LIN {X 0,Y 573.266,Z 445.075,A -85,B 0,C 180,E1 -2313.81,E2 -2313.81} C_VEL
LIN {X 0,Y 573.234,Z 445.082,A -85,B 0,C 180,E1 -2316.135,E2 -2316.135} C_VEL
LIN {X 0,Y 573.254,Z 445.079,A -85,B 0,C 180,E1 -2319.174,E2 -2319.174} C_VEL
LIN {X 0,Y 573.23,Z 445.081,A -85,B 0,C 180,E1 -2321.412,E2 -2321.412} C_VEL
LIN {X 0,Y 573.254,Z 445.077,A -85,B 0,C 180,E1 -2323.622,E2 -2323.622} C_VEL
LIN {X 0,Y 573.276,Z 445.079,A -85,B 0,C 180,E1 -2325.807,E2 -2325.807} C_VEL
LIN {X 0,Y 573.266,Z 445.08,A -85,B 0,C 180,E1 -2328.745,E2 -2328.745} C_VEL
LIN {X 0,Y 573.287,Z 445.073,A -85,B 0,C 180,E1 -2331.541,E2 -2331.541} C_VEL
LIN {X 0,Y 573.292,Z 445.072,A -85,B 0,C 180,E1 -2334.372,E2 -2334.372} C_VEL
LIN {X 0,Y 573.308,Z 445.071,A -85,B 0,C 180,E1 -2337.893,E2 -2337.893} C_VEL
LIN {X 0,Y 573.337,Z 445.066,A -85,B 0,C 180,E1 -2340.702,E2 -2340.702} C_VEL
LIN {X 0,Y 573.234,Z 445.079,A -85,B 0,C 180,E1 -2343.515,E2 -2343.515} C_VEL
LIN {X 0,Y 573.291,Z 445.073,A -85,B 0,C 180,E1 -2345.628,E2 -2345.628} C_VEL
LIN {X 0,Y 573.292,Z 445.072,A -85,B 0,C 180,E1 -2348.46,E2 -2348.46} C_VEL
LIN {X 0,Y 573.275,Z 445.073,A -85,B 0,C 180,E1 -2351.312,E2 -2351.312} C_VEL
LIN {X 0,Y 573.285,Z 445.073,A -85,B 0,C 180,E1 -2354.425,E2 -2354.425} C_VEL
LIN {X 0,Y 573.262,Z 445.079,A -85,B 0,C 180,E1 -2357.112,E2 -2357.112} C_VEL
LIN {X 0,Y 573.255,Z 445.082,A -85,B 0,C 180,E1 -2360.077,E2 -2360.077} C_VEL
LIN {X 0,Y 573.238,Z 445.084,A -85,B 0,C 180,E1 -2363.1,E2 -2363.1} C_VEL
LIN {X 0,Y 573.253,Z 445.079,A -85,B 0,C 180,E1 -2364.389,E2 -2364.389} C_VEL
LIN {X 0,Y 572.625,Z 445.161,A -85,B 0,C 180,E1 -2364.976,E2 -2364.976} C_VEL
LIN {X 0,Y 569.778,Z 445.516,A -85,B 0,C 180,E1 -2365.927,E2 -2365.927} C_VEL
LIN {X 0,Y 567.345,Z 445.816,A -85,B 0,C 180,E1 -2366.692,E2 -2366.692} C_VEL
LIN {X 0,Y 566.296,Z 445.944,A -85,B 0,C 180,E1 -2367.284,E2 -2367.284} C_VEL
LIN {X 0,Y 566.21,Z 445.954,A -85,B 0,C 180,E1 -2367.484,E2 -2367.484} C_VEL
LIN {X 0,Y 566.205,Z 445.957,A -85,B 0,C 180,E1 -2369.769,E2 -2369.769} C_VEL
LIN {X 0,Y 566.209,Z 445.959,A -85,B 0,C 180,E1 -2372.43,E2 -2372.43} C_VEL
LIN {X 0,Y 566.205,Z 445.955,A -85,B 0,C 180,E1 -2374.993,E2 -2374.993} C_VEL
LIN {X 0,Y 566.2,Z 445.958,A -85,B 0,C 180,E1 -2377.461,E2 -2377.461} C_VEL
LIN {X 0,Y 566.21,Z 445.958,A -85,B 0,C 180,E1 -2380.199,E2 -2380.199} C_VEL
LIN {X 0,Y 566.209,Z 445.956,A -85,B 0,C 180,E1 -2383.054,E2 -2383.054} C_VEL
LIN {X 0,Y 566.202,Z 445.956,A -85,B 0,C 180,E1 -2386.049,E2 -2386.049} C_VEL
LIN {X 0,Y 566.207,Z 445.955,A -85,B 0,C 180,E1 -2389.215,E2 -2389.215} C_VEL
LIN {X 0,Y 566.19,Z 445.958,A -85,B 0,C 180,E1 -2391.637,E2 -2391.637} C_VEL
LIN {X 0,Y 566.196,Z 445.961,A -85,B 0,C 180,E1 -2394.31,E2 -2394.31} C_VEL
LIN {X 0,Y 566.224,Z 445.952,A -85,B 0,C 180,E1 -2396.898,E2 -2396.898} C_VEL
LIN {X 0,Y 566.184,Z 445.959,A -85,B 0,C 180,E1 -2399.407,E2 -2399.407} C_VEL
LIN {X 0,Y 566.199,Z 445.957,A -85,B 0,C 180,E1 -2401.857,E2 -2401.857} C_VEL
LIN {X 0,Y 566.218,Z 445.954,A -85,B 0,C 180,E1 -2404.251,E2 -2404.251} C_VEL
LIN {X 0,Y 566.178,Z 445.963,A -85,B 0,C 180,E1 -2406.718,E2 -2406.718} C_VEL
LIN {X 0,Y 566.211,Z 445.956,A -85,B 0,C 180,E1 -2409.663,E2 -2409.663} C_VEL
LIN {X 0,Y 566.204,Z 445.956,A -85,B 0,C 180,E1 -2412.669,E2 -2412.669} C_VEL
LIN {X 0,Y 566.24,Z 445.95,A -85,B 0,C 180,E1 -2415.627,E2 -2415.627} C_VEL
LIN {X 0,Y 566.241,Z 445.95,A -85,B 0,C 180,E1 -2418.675,E2 -2418.675} C_VEL
LIN {X 0,Y 566.233,Z 445.952,A -85,B 0,C 180,E1 -2421.434,E2 -2421.434} C_VEL
LIN {X 0,Y 566.257,Z 445.95,A -85,B 0,C 180,E1 -2424.302,E2 -2424.302} C_VEL
LIN {X 0,Y 566.288,Z 445.944,A -85,B 0,C 180,E1 -2427.866,E2 -2427.866} C_VEL
LIN {X 0,Y 566.304,Z 445.943,A -85,B 0,C 180,E1 -2430.711,E2 -2430.711} C_VEL
LIN {X 0,Y 566.273,Z 445.947,A -85,B 0,C 180,E1 -2432.846,E2 -2432.846} C_VEL
LIN {X 0,Y 566.263,Z 445.947,A -85,B 0,C 180,E1 -2435.698,E2 -2435.698} C_VEL
LIN {X 0,Y 566.212,Z 445.954,A -85,B 0,C 180,E1 -2438.566,E2 -2438.566} C_VEL
LIN {X 0,Y 566.248,Z 445.952,A -85,B 0,C 180,E1 -2441.454,E2 -2441.454} C_VEL
LIN {X 0,Y 566.241,Z 445.953,A -85,B 0,C 180,E1 -2444.507,E2 -2444.507} C_VEL
LIN {X 0,Y 566.205,Z 445.959,A -85,B 0,C 180,E1 -2447.332,E2 -2447.332} C_VEL
LIN {X 0,Y 566.214,Z 445.957,A -85,B 0,C 180,E1 -2450.337,E2 -2450.337} C_VEL
LIN {X 0,Y 566.178,Z 445.959,A -85,B 0,C 180,E1 -2453.282,E2 -2453.282} C_VEL
LIN {X 0,Y 566.219,Z 445.953,A -85,B 0,C 180,E1 -2455.749,E2 -2455.749} C_VEL
LIN {X 0,Y 566.208,Z 445.959,A -85,B 0,C 180,E1 -2458.202,E2 -2458.202} C_VEL
LIN {X 0,Y 566.196,Z 445.957,A -85,B 0,C 180,E1 -2461.076,E2 -2461.076} C_VEL
LIN {X 0,Y 566.217,Z 445.953,A -85,B 0,C 180,E1 -2463.734,E2 -2463.734} C_VEL
LIN {X 0,Y 566.204,Z 445.955,A -85,B 0,C 180,E1 -2466.57,E2 -2466.57} C_VEL
LIN {X 0,Y 566.225,Z 445.953,A -85,B 0,C 180,E1 -2469.686,E2 -2469.686} C_VEL
LIN {X 0,Y 566.216,Z 445.956,A -85,B 0,C 180,E1 -2472.087,E2 -2472.087} C_VEL
LIN {X 0,Y 566.174,Z 445.959,A -85,B 0,C 180,E1 -2475.036,E2 -2475.036} C_VEL
LIN {X 0,Y 566.223,Z 445.954,A -85,B 0,C 180,E1 -2478.136,E2 -2478.136} C_VEL
LIN {X 0,Y 566.216,Z 445.953,A -85,B 0,C 180,E1 -2480.726,E2 -2480.726} C_VEL
LIN {X 0,Y 566.197,Z 445.96,A -85,B 0,C 180,E1 -2483.429,E2 -2483.429} C_VEL
LIN {X 0,Y 566.027,Z 445.982,A -85,B 0,C 180,E1 -2486.031,E2 -2486.031} C_VEL
LIN {X 0,Y 565.995,Z 446.653,A -85,B 0,C 180,E1 -2486.883,E2 -2486.883} C_VEL
LIN {X 0,Y 565.971,Z 449.517,A -85,B 0,C 180,E1 -2489.394,E2 -2489.394} C_VEL
LIN {X 0,Y 565.965,Z 452.327,A -85,B 0,C 180,E1 -2491.844,E2 -2491.844} C_VEL
LIN {X 0,Y 565.945,Z 455.14,A -85,B 0,C 180,E1 -2494.238,E2 -2494.238} C_VEL
LIN {X 0,Y 565.898,Z 458.02,A -85,B 0,C 180,E1 -2496.784,E2 -2496.784} C_VEL
LIN {X 0,Y 565.884,Z 461.612,A -85,B 0,C 180,E1 -2499.65,E2 -2499.65} C_VEL
LIN {X 0,Y 565.864,Z 465.455,A -85,B 0,C 180,E1 -2502.658,E2 -2502.658} C_VEL
LIN {X 0,Y 565.889,Z 469.316,A -85,B 0,C 180,E1 -2505.631,E2 -2505.631} C_VEL
LIN {X 0,Y 565.897,Z 471.671,A -85,B 0,C 180,E1 -2507.424,E2 -2507.424} C_VEL
LIN {X 0,Y 566.89,Z 479.272,A -85,B 0,C 180,E1 -2507.629,E2 -2507.629} C_VEL
LIN {X 0,Y 566.784,Z 491.774,A -85,B 0,C 180,E1 -2508.013,E2 -2508.013} C_VEL
LIN {X 0,Y 566.661,Z 504.296,A -85,B 0,C 180,E1 -2508.554,E2 -2508.554} C_VEL
LIN {X 0,Y 566.544,Z 515.576,A -85,B 0,C 180,E1 -2509.192,E2 -2509.192} C_VEL
LIN {X 0,Y 566.342,Z 526.839,A -85,B 0,C 180,E1 -2509.995,E2 -2509.995} C_VEL
LIN {X 0,Y 566.238,Z 536.889,A -85,B 0,C 180,E1 -2510.895,E2 -2510.895} C_VEL
LIN {X 0,Y 566.113,Z 546.59,A -85,B 0,C 180,E1 -2511.971,E2 -2511.971} C_VEL
LIN {X 0,Y 566.05,Z 553.158,A -85,B 0,C 180,E1 -2512.868,E2 -2512.868} C_VEL
LIN {X 0,Y 566.003,Z 559.627,A -85,B 0,C 180,E1 -2513.941,E2 -2513.941} C_VEL
LIN {X 0,Y 565.878,Z 564.764,A -85,B 0,C 180,E1 -2515.012,E2 -2515.012} C_VEL
LIN {X 0,Y 565.926,Z 568.753,A -85,B 0,C 180,E1 -2516.083,E2 -2516.083} C_VEL
LIN {X 0,Y 565.878,Z 571.701,A -85,B 0,C 180,E1 -2517.152,E2 -2517.152} C_VEL
LIN {X 0,Y 565.839,Z 573.128,A -85,B 0,C 180,E1 -2517.864,E2 -2517.864} C_VEL
LIN {X 0,Y 565.842,Z 574.756,A -85,B 0,C 180,E1 -2519.288,E2 -2519.288} C_VEL
LIN {X 0,Y 565.839,Z 574.996,A -85,B 0,C 180,E1 -2520,E2 -2520} C_VEL
LIN {X 0,Y 565.841,Z 574.815,A -85,B 0,C 180,E1 -2520.712,E2 -2520.712} C_VEL
LIN {X 0,Y 565.838,Z 573.269,A -85,B 0,C 180,E1 -2522.135,E2 -2522.135} C_VEL
LIN {X 0,Y 565.878,Z 571.908,A -85,B 0,C 180,E1 -2522.847,E2 -2522.847} C_VEL
LIN {X 0,Y 565.926,Z 569.03,A -85,B 0,C 180,E1 -2523.916,E2 -2523.916} C_VEL
LIN {X 0,Y 565.878,Z 565.13,A -85,B 0,C 180,E1 -2524.987,E2 -2524.987} C_VEL
LIN {X 0,Y 565.994,Z 560.097,A -85,B 0,C 180,E1 -2526.058,E2 -2526.058} C_VEL
LIN {X 0,Y 566.031,Z 553.773,A -85,B 0,C 180,E1 -2527.132,E2 -2527.132} C_VEL
LIN {X 0,Y 566.128,Z 545.851,A -85,B 0,C 180,E1 -2528.208,E2 -2528.208} C_VEL
LIN {X 0,Y 566.249,Z 536,A -85,B 0,C 180,E1 -2529.285,E2 -2529.285} C_VEL
LIN {X 0,Y 566.412,Z 525.679,A -85,B 0,C 180,E1 -2530.184,E2 -2530.184} C_VEL
LIN {X 0,Y 566.525,Z 514.433,A -85,B 0,C 180,E1 -2530.97,E2 -2530.97} C_VEL
LIN {X 0,Y 566.684,Z 502.858,A -85,B 0,C 180,E1 -2531.608,E2 -2531.608} C_VEL
LIN {X 0,Y 566.783,Z 490.466,A -85,B 0,C 180,E1 -2532.124,E2 -2532.124} C_VEL
LIN {X 0,Y 566.817,Z 477.42,A -85,B 0,C 180,E1 -2532.509,E2 -2532.509} C_VEL
LIN {X 0,Y 565.899,Z 471.67,A -85,B 0,C 180,E1 -2532.666,E2 -2532.666} C_VEL
LIN {X 0,Y 565.857,Z 468.455,A -85,B 0,C 180,E1 -2535.119,E2 -2535.119} C_VEL
LIN {X 0,Y 565.863,Z 465.571,A -85,B 0,C 180,E1 -2537.342,E2 -2537.342} C_VEL
LIN {X 0,Y 565.884,Z 461.726,A -85,B 0,C 180,E1 -2540.35,E2 -2540.35} C_VEL
LIN {X 0,Y 565.898,Z 458.134,A -85,B 0,C 180,E1 -2543.216,E2 -2543.216} C_VEL
LIN {X 0,Y 565.962,Z 455.534,A -85,B 0,C 180,E1 -2545.761,E2 -2545.761} C_VEL
LIN {X 0,Y 566.028,Z 453.112,A -85,B 0,C 180,E1 -2548.168,E2 -2548.168} C_VEL
LIN {X 0,Y 566.078,Z 450.089,A -85,B 0,C 180,E1 -2551.057,E2 -2551.057} C_VEL
LIN {X 0,Y 566.109,Z 447.052,A -85,B 0,C 180,E1 -2553.963,E2 -2553.963} C_VEL
LIN {X 0,Y 566.117,Z 446.004,A -85,B 0,C 180,E1 -2554.98,E2 -2554.98} C_VEL
LIN {X 0,Y 566.2,Z 445.959,A -85,B 0,C 180,E1 -2557.461,E2 -2557.461} C_VEL
LIN {X 0,Y 566.21,Z 445.96,A -85,B 0,C 180,E1 -2560.199,E2 -2560.199} C_VEL
LIN {X 0,Y 566.209,Z 445.958,A -85,B 0,C 180,E1 -2563.054,E2 -2563.054} C_VEL
LIN {X 0,Y 566.201,Z 445.96,A -85,B 0,C 180,E1 -2566.049,E2 -2566.049} C_VEL
LIN {X 0,Y 566.224,Z 445.956,A -85,B 0,C 180,E1 -2569.212,E2 -2569.212} C_VEL
LIN {X 0,Y 566.209,Z 445.959,A -85,B 0,C 180,E1 -2572.091,E2 -2572.091} C_VEL
LIN {X 0,Y 566.225,Z 446.171,A -85,B 0,C 180,E1 -2572.596,E2 -2572.596} C_VEL
LIN {X 0,Y 566.879,Z 450.21,A -85,B 0,C 180,E1 -2574.36,E2 -2574.36} C_VEL
LIN {X 0,Y 566.688,Z 456.223,A -85,B 0,C 180,E1 -2576.553,E2 -2576.553} C_VEL
LIN {X 0,Y 566.562,Z 463.236,A -85,B 0,C 180,E1 -2578.862,E2 -2578.862} C_VEL
LIN {X 0,Y 566.448,Z 471.711,A -85,B 0,C 180,E1 -2581.443,E2 -2581.443} C_VEL
LIN {X 0,Y 566.425,Z 480.069,A -85,B 0,C 180,E1 -2583.866,E2 -2583.866} C_VEL
LIN {X 0,Y 566.361,Z 488.309,A -85,B 0,C 180,E1 -2586.216,E2 -2586.216} C_VEL
LIN {X 0,Y 566.245,Z 497.576,A -85,B 0,C 180,E1 -2588.904,E2 -2588.904} C_VEL
LIN {X 0,Y 566.167,Z 506.844,A -85,B 0,C 180,E1 -2591.546,E2 -2591.546} C_VEL
LIN {X 0,Y 566.092,Z 517.435,A -85,B 0,C 180,E1 -2594.519,E2 -2594.519} C_VEL
LIN {X 0,Y 566.033,Z 527.53,A -85,B 0,C 180,E1 -2597.314,E2 -2597.314} C_VEL
LIN {X 0,Y 566.942,Z 534.363,A -85,B 0,C 180,E1 -2597.471,E2 -2597.471} C_VEL
LIN {X 0,Y 566.829,Z 546.495,A -85,B 0,C 180,E1 -2597.786,E2 -2597.786} C_VEL
LIN {X 0,Y 566.719,Z 558.314,A -85,B 0,C 180,E1 -2598.229,E2 -2598.229} C_VEL
LIN {X 0,Y 566.572,Z 570.724,A -85,B 0,C 180,E1 -2598.854,E2 -2598.854} C_VEL
LIN {X 0,Y 566.419,Z 581.48,A -85,B 0,C 180,E1 -2599.545,E2 -2599.545} C_VEL
LIN {X 0,Y 566.301,Z 591.646,A -85,B 0,C 180,E1 -2600.355,E2 -2600.355} C_VEL
LIN {X 0,Y 566.166,Z 600.786,A -85,B 0,C 180,E1 -2601.253,E2 -2601.253} C_VEL
LIN {X 0,Y 566.08,Z 609.689,A -85,B 0,C 180,E1 -2602.33,E2 -2602.33} C_VEL
LIN {X 0,Y 565.967,Z 616.955,A -85,B 0,C 180,E1 -2603.422,E2 -2603.422} C_VEL
LIN {X 0,Y 566.004,Z 621.679,A -85,B 0,C 180,E1 -2604.299,E2 -2604.299} C_VEL
LIN {X 0,Y 565.933,Z 626.372,A -85,B 0,C 180,E1 -2605.37,E2 -2605.37} C_VEL
LIN {X 0,Y 565.927,Z 629.957,A -85,B 0,C 180,E1 -2606.44,E2 -2606.44} C_VEL
LIN {X 0,Y 565.878,Z 631.808,A -85,B 0,C 180,E1 -2607.152,E2 -2607.152} C_VEL
LIN {X 0,Y 565.846,Z 634.186,A -85,B 0,C 180,E1 -2608.577,E2 -2608.577} C_VEL
LIN {X 0,Y 565.839,Z 635,A -85,B 0,C 180,E1 -2610,E2 -2610} C_VEL
LIN {X 0,Y 565.846,Z 634.186,A -85,B 0,C 180,E1 -2611.423,E2 -2611.423} C_VEL
LIN {X 0,Y 565.878,Z 631.81,A -85,B 0,C 180,E1 -2612.847,E2 -2612.847} C_VEL
LIN {X 0,Y 565.926,Z 628.896,A -85,B 0,C 180,E1 -2613.916,E2 -2613.916} C_VEL
LIN {X 0,Y 565.878,Z 624.949,A -85,B 0,C 180,E1 -2614.987,E2 -2614.987} C_VEL
LIN {X 0,Y 566.002,Z 619.867,A -85,B 0,C 180,E1 -2616.058,E2 -2616.058} C_VEL
LIN {X 0,Y 566.04,Z 613.469,A -85,B 0,C 180,E1 -2617.132,E2 -2617.132} C_VEL
LIN {X 0,Y 566.133,Z 605.479,A -85,B 0,C 180,E1 -2618.208,E2 -2618.208} C_VEL
LIN {X 0,Y 566.229,Z 597.336,A -85,B 0,C 180,E1 -2619.105,E2 -2619.105} C_VEL
LIN {X 0,Y 566.342,Z 587.401,A -85,B 0,C 180,E1 -2620.005,E2 -2620.005} C_VEL
LIN {X 0,Y 566.534,Z 576.299,A -85,B 0,C 180,E1 -2620.807,E2 -2620.807} C_VEL
LIN {X 0,Y 566.612,Z 565.178,A -85,B 0,C 180,E1 -2621.447,E2 -2621.447} C_VEL
LIN {X 0,Y 566.756,Z 552.985,A -85,B 0,C 180,E1 -2621.988,E2 -2621.988} C_VEL
LIN {X 0,Y 566.881,Z 540.178,A -85,B 0,C 180,E1 -2622.394,E2 -2622.394} C_VEL
LIN {X 0,Y 566.716,Z 531.802,A -85,B 0,C 180,E1 -2622.585,E2 -2622.585} C_VEL
LIN {X 0,Y 566.033,Z 527.53,A -85,B 0,C 180,E1 -2622.686,E2 -2622.686} C_VEL
LIN {X 0,Y 566.091,Z 517.436,A -85,B 0,C 180,E1 -2625.481,E2 -2625.481} C_VEL
LIN {X 0,Y 566.167,Z 506.844,A -85,B 0,C 180,E1 -2628.454,E2 -2628.454} C_VEL
LIN {X 0,Y 566.245,Z 497.577,A -85,B 0,C 180,E1 -2631.096,E2 -2631.096} C_VEL
LIN {X 0,Y 566.362,Z 488.31,A -85,B 0,C 180,E1 -2633.784,E2 -2633.784} C_VEL
LIN {X 0,Y 566.473,Z 478.959,A -85,B 0,C 180,E1 -2636.528,E2 -2636.528} C_VEL
LIN {X 0,Y 566.558,Z 469.563,A -85,B 0,C 180,E1 -2639.34,E2 -2639.34} C_VEL
LIN {X 0,Y 566.669,Z 461.593,A -85,B 0,C 180,E1 -2641.81,E2 -2641.81} C_VEL
LIN {X 0,Y 566.865,Z 453.765,A -85,B 0,C 180,E1 -2644.341,E2 -2644.341} C_VEL
LIN {X 0,Y 566.815,Z 449.857,A -85,B 0,C 180,E1 -2645.645,E2 -2645.645} C_VEL
LIN {X 0,Y 566.221,Z 445.957,A -85,B 0,C 180,E1 -2647.061,E2 -2647.061} C_VEL
LIN {X 0,Y 566.215,Z 445.958,A -85,B 0,C 180,E1 -2649.685,E2 -2649.685} C_VEL
LIN {X 0,Y 566.192,Z 445.957,A -85,B 0,C 180,E1 -2652.089,E2 -2652.089} C_VEL
LIN {X 0,Y 566.176,Z 445.959,A -85,B 0,C 180,E1 -2655.036,E2 -2655.036} C_VEL
LIN {X 0,Y 566.217,Z 445.956,A -85,B 0,C 180,E1 -2657.913,E2 -2657.913} C_VEL
LIN {X 0,Y 566.214,Z 445.959,A -85,B 0,C 180,E1 -2660.726,E2 -2660.726} C_VEL
LIN {X 0,Y 566.188,Z 445.962,A -85,B 0,C 180,E1 -2663.788,E2 -2663.788} C_VEL
LIN {X 0,Y 566.214,Z 445.953,A -85,B 0,C 180,E1 -2666.266,E2 -2666.266} C_VEL
LIN {X 0,Y 566.193,Z 445.958,A -85,B 0,C 180,E1 -2668.924,E2 -2668.924} C_VEL
LIN {X 0,Y 566.214,Z 445.958,A -85,B 0,C 180,E1 -2671.857,E2 -2671.857} C_VEL
LIN {X 0,Y 566.216,Z 445.954,A -85,B 0,C 180,E1 -2674.251,E2 -2674.251} C_VEL
LIN {X 0,Y 566.175,Z 445.96,A -85,B 0,C 180,E1 -2676.718,E2 -2676.718} C_VEL
LIN {X 0,Y 566.217,Z 445.957,A -85,B 0,C 180,E1 -2679.663,E2 -2679.663} C_VEL
LIN {X 0,Y 566.202,Z 445.96,A -85,B 0,C 180,E1 -2682.668,E2 -2682.668} C_VEL
LIN {X 0,Y 566.237,Z 445.955,A -85,B 0,C 180,E1 -2685.627,E2 -2685.627} C_VEL
LIN {X 0,Y 566.237,Z 445.954,A -85,B 0,C 180,E1 -2688.675,E2 -2688.675} C_VEL
LIN {X 0,Y 566.23,Z 445.952,A -85,B 0,C 180,E1 -2691.434,E2 -2691.434} C_VEL
LIN {X 0,Y 566.26,Z 445.948,A -85,B 0,C 180,E1 -2694.302,E2 -2694.302} C_VEL
LIN {X 0,Y 566.28,Z 445.947,A -85,B 0,C 180,E1 -2697.866,E2 -2697.866} C_VEL
LIN {X 0,Y 566.307,Z 445.942,A -85,B 0,C 180,E1 -2700.711,E2 -2700.711} C_VEL
LIN {X 0,Y 566.278,Z 445.951,A -85,B 0,C 180,E1 -2702.846,E2 -2702.846} C_VEL
LIN {X 0,Y 566.26,Z 445.95,A -85,B 0,C 180,E1 -2705.698,E2 -2705.698} C_VEL
LIN {X 0,Y 566.236,Z 445.951,A -85,B 0,C 180,E1 -2708.566,E2 -2708.566} C_VEL
LIN {X 0,Y 566.245,Z 445.949,A -85,B 0,C 180,E1 -2711.454,E2 -2711.454} C_VEL
LIN {X 0,Y 566.238,Z 445.951,A -85,B 0,C 180,E1 -2714.507,E2 -2714.507} C_VEL
LIN {X 0,Y 566.203,Z 445.956,A -85,B 0,C 180,E1 -2717.332,E2 -2717.332} C_VEL
LIN {X 0,Y 566.217,Z 445.956,A -85,B 0,C 180,E1 -2720.337,E2 -2720.337} C_VEL
LIN {X 0,Y 566.176,Z 445.963,A -85,B 0,C 180,E1 -2723.282,E2 -2723.282} C_VEL
LIN {X 0,Y 566.216,Z 445.953,A -85,B 0,C 180,E1 -2725.749,E2 -2725.749} C_VEL
LIN {X 0,Y 566.21,Z 445.954,A -85,B 0,C 180,E1 -2727.484,E2 -2727.484} C_VEL
LIN {X 0,Y 565.538,Z 446.041,A -85,B 0,C 180,E1 -2728.078,E2 -2728.078} C_VEL
LIN {X 0,Y 562.671,Z 446.397,A -85,B 0,C 180,E1 -2729.041,E2 -2729.041} C_VEL
LIN {X 0,Y 560.254,Z 446.698,A -85,B 0,C 180,E1 -2729.817,E2 -2729.817} C_VEL
LIN {X 0,Y 559.224,Z 446.825,A -85,B 0,C 180,E1 -2730.415,E2 -2730.415} C_VEL
LIN {X 0,Y 559.143,Z 446.835,A -85,B 0,C 180,E1 -2730.618,E2 -2730.618} C_VEL
LIN {X 0,Y 559.168,Z 446.831,A -85,B 0,C 180,E1 -2733.575,E2 -2733.575} C_VEL
LIN {X 0,Y 559.171,Z 446.831,A -85,B 0,C 180,E1 -2736.448,E2 -2736.448} C_VEL
LIN {X 0,Y 559.177,Z 446.834,A -85,B 0,C 180,E1 -2738.934,E2 -2738.934} C_VEL
LIN {X 0,Y 559.181,Z 446.833,A -85,B 0,C 180,E1 -2742.138,E2 -2742.138} C_VEL
LIN {X 0,Y 559.145,Z 446.837,A -85,B 0,C 180,E1 -2744.739,E2 -2744.739} C_VEL
LIN {X 0,Y 559.161,Z 446.832,A -85,B 0,C 180,E1 -2747.256,E2 -2747.256} C_VEL
LIN {X 0,Y 559.184,Z 446.831,A -85,B 0,C 180,E1 -2750.135,E2 -2750.135} C_VEL
LIN {X 0,Y 559.148,Z 446.838,A -85,B 0,C 180,E1 -2752.892,E2 -2752.892} C_VEL
LIN {X 0,Y 559.172,Z 446.835,A -85,B 0,C 180,E1 -2756.051,E2 -2756.051} C_VEL
LIN {X 0,Y 559.159,Z 446.837,A -85,B 0,C 180,E1 -2758.981,E2 -2758.981} C_VEL
LIN {X 0,Y 559.173,Z 446.831,A -85,B 0,C 180,E1 -2761.619,E2 -2761.619} C_VEL
LIN {X 0,Y 559.181,Z 446.83,A -85,B 0,C 180,E1 -2764.702,E2 -2764.702} C_VEL
LIN {X 0,Y 559.145,Z 446.835,A -85,B 0,C 180,E1 -2767.847,E2 -2767.847} C_VEL
LIN {X 0,Y 559.197,Z 446.828,A -85,B 0,C 180,E1 -2770.494,E2 -2770.494} C_VEL
LIN {X 0,Y 559.184,Z 446.834,A -85,B 0,C 180,E1 -2773.198,E2 -2773.198} C_VEL
LIN {X 0,Y 559.177,Z 446.836,A -85,B 0,C 180,E1 -2776.184,E2 -2776.184} C_VEL
LIN {X 0,Y 559.201,Z 446.831,A -85,B 0,C 180,E1 -2779.134,E2 -2779.134} C_VEL
LIN {X 0,Y 559.209,Z 446.828,A -85,B 0,C 180,E1 -2782.054,E2 -2782.054} C_VEL
LIN {X 0,Y 559.254,Z 446.82,A -85,B 0,C 180,E1 -2784.953,E2 -2784.953} C_VEL
LIN {X 0,Y 559.259,Z 446.82,A -85,B 0,C 180,E1 -2787.84,E2 -2787.84} C_VEL
LIN {X 0,Y 559.275,Z 446.818,A -85,B 0,C 180,E1 -2790.72,E2 -2790.72} C_VEL
LIN {X 0,Y 559.24,Z 446.823,A -85,B 0,C 180,E1 -2792.881,E2 -2792.881} C_VEL
LIN {X 0,Y 559.233,Z 446.823,A -85,B 0,C 180,E1 -2795.77,E2 -2795.77} C_VEL
LIN {X 0,Y 559.176,Z 446.83,A -85,B 0,C 180,E1 -2798.675,E2 -2798.675} C_VEL
LIN {X 0,Y 559.212,Z 446.827,A -85,B 0,C 180,E1 -2801.6,E2 -2801.6} C_VEL
LIN {X 0,Y 559.206,Z 446.828,A -85,B 0,C 180,E1 -2804.596,E2 -2804.596} C_VEL
LIN {X 0,Y 559.164,Z 446.836,A -85,B 0,C 180,E1 -2807.557,E2 -2807.557} C_VEL
LIN {X 0,Y 559.172,Z 446.831,A -85,B 0,C 180,E1 -2809.838,E2 -2809.838} C_VEL
LIN {X 0,Y 559.146,Z 446.838,A -85,B 0,C 180,E1 -2812.153,E2 -2812.153} C_VEL
LIN {X 0,Y 559.182,Z 446.835,A -85,B 0,C 180,E1 -2815.298,E2 -2815.298} C_VEL
LIN {X 0,Y 559.161,Z 446.833,A -85,B 0,C 180,E1 -2817.713,E2 -2817.713} C_VEL
LIN {X 0,Y 559.159,Z 446.834,A -85,B 0,C 180,E1 -2820.183,E2 -2820.183} C_VEL
LIN {X 0,Y 559.161,Z 446.835,A -85,B 0,C 180,E1 -2822.715,E2 -2822.715} C_VEL
LIN {X 0,Y 559.134,Z 446.835,A -85,B 0,C 180,E1 -2825.324,E2 -2825.324} C_VEL
LIN {X 0,Y 559.138,Z 446.837,A -85,B 0,C 180,E1 -2828.017,E2 -2828.017} C_VEL
LIN {X 0,Y 559.162,Z 446.837,A -85,B 0,C 180,E1 -2830.812,E2 -2830.812} C_VEL
LIN {X 0,Y 559.15,Z 446.833,A -85,B 0,C 180,E1 -2833.196,E2 -2833.196} C_VEL
LIN {X 0,Y 559.146,Z 446.834,A -85,B 0,C 180,E1 -2836.266,E2 -2836.266} C_VEL
LIN {X 0,Y 559.173,Z 446.833,A -85,B 0,C 180,E1 -2838.948,E2 -2838.948} C_VEL
LIN {X 0,Y 559.177,Z 446.83,A -85,B 0,C 180,E1 -2841.192,E2 -2841.192} C_VEL
LIN {X 0,Y 559.128,Z 446.837,A -85,B 0,C 180,E1 -2843.788,E2 -2843.788} C_VEL
LIN {X 0,Y 558.929,Z 446.866,A -85,B 0,C 180,E1 -2846.409,E2 -2846.409} C_VEL
LIN {X 0,Y 558.925,Z 449.618,A -85,B 0,C 180,E1 -2848.966,E2 -2848.966} C_VEL
LIN {X 0,Y 558.88,Z 452.694,A -85,B 0,C 180,E1 -2851.674,E2 -2851.674} C_VEL
LIN {X 0,Y 558.863,Z 455.235,A -85,B 0,C 180,E1 -2853.887,E2 -2853.887} C_VEL
LIN {X 0,Y 558.831,Z 458.402,A -85,B 0,C 180,E1 -2856.646,E2 -2856.646} C_VEL
LIN {X 0,Y 558.79,Z 461.613,A -85,B 0,C 180,E1 -2859.38,E2 -2859.38} C_VEL
LIN {X 0,Y 558.765,Z 464.495,A -85,B 0,C 180,E1 -2861.673,E2 -2861.673} C_VEL
LIN {X 0,Y 558.773,Z 467.378,A -85,B 0,C 180,E1 -2863.936,E2 -2863.936} C_VEL
LIN {X 0,Y 558.782,Z 470.26,A -85,B 0,C 180,E1 -2866.174,E2 -2866.174} C_VEL
LIN {X 0,Y 558.804,Z 471.672,A -85,B 0,C 180,E1 -2867.262,E2 -2867.262} C_VEL
LIN {X 0,Y 559.966,Z 480.209,A -85,B 0,C 180,E1 -2867.496,E2 -2867.496} C_VEL
LIN {X 0,Y 559.853,Z 492.293,A -85,B 0,C 180,E1 -2867.88,E2 -2867.88} C_VEL
LIN {X 0,Y 559.688,Z 504.306,A -85,B 0,C 180,E1 -2868.41,E2 -2868.41} C_VEL
LIN {X 0,Y 559.566,Z 515.653,A -85,B 0,C 180,E1 -2869.06,E2 -2869.06} C_VEL
LIN {X 0,Y 559.357,Z 526.848,A -85,B 0,C 180,E1 -2869.869,E2 -2869.869} C_VEL
LIN {X 0,Y 559.211,Z 536.894,A -85,B 0,C 180,E1 -2870.779,E2 -2870.779} C_VEL
LIN {X 0,Y 559.051,Z 546.594,A -85,B 0,C 180,E1 -2871.869,E2 -2871.869} C_VEL
LIN {X 0,Y 558.971,Z 554.454,A -85,B 0,C 180,E1 -2872.977,E2 -2872.977} C_VEL
LIN {X 0,Y 558.936,Z 561.454,A -85,B 0,C 180,E1 -2874.227,E2 -2874.227} C_VEL
LIN {X 0,Y 558.826,Z 566.194,A -85,B 0,C 180,E1 -2875.311,E2 -2875.311} C_VEL
LIN {X 0,Y 558.837,Z 569.827,A -85,B 0,C 180,E1 -2876.395,E2 -2876.395} C_VEL
LIN {X 0,Y 558.8,Z 571.703,A -85,B 0,C 180,E1 -2877.116,E2 -2877.116} C_VEL
LIN {X 0,Y 558.745,Z 573.128,A -85,B 0,C 180,E1 -2877.837,E2 -2877.837} C_VEL
LIN {X 0,Y 558.742,Z 574.756,A -85,B 0,C 180,E1 -2879.279,E2 -2879.279} C_VEL
LIN {X 0,Y 558.74,Z 574.996,A -85,B 0,C 180,E1 -2880,E2 -2880} C_VEL
LIN {X 0,Y 558.741,Z 574.814,A -85,B 0,C 180,E1 -2880.721,E2 -2880.721} C_VEL
LIN {X 0,Y 558.744,Z 573.267,A -85,B 0,C 180,E1 -2882.162,E2 -2882.162} C_VEL
LIN {X 0,Y 558.8,Z 571.906,A -85,B 0,C 180,E1 -2882.884,E2 -2882.884} C_VEL
LIN {X 0,Y 558.844,Z 569.028,A -85,B 0,C 180,E1 -2883.966,E2 -2883.966} C_VEL
LIN {X 0,Y 558.798,Z 565.127,A -85,B 0,C 180,E1 -2885.051,E2 -2885.051} C_VEL
LIN {X 0,Y 558.913,Z 560.094,A -85,B 0,C 180,E1 -2886.136,E2 -2886.136} C_VEL
LIN {X 0,Y 558.972,Z 553.769,A -85,B 0,C 180,E1 -2887.223,E2 -2887.223} C_VEL
LIN {X 0,Y 559.091,Z 545.846,A -85,B 0,C 180,E1 -2888.312,E2 -2888.312} C_VEL
LIN {X 0,Y 559.223,Z 535.994,A -85,B 0,C 180,E1 -2889.403,E2 -2889.403} C_VEL
LIN {X 0,Y 559.399,Z 525.673,A -85,B 0,C 180,E1 -2890.313,E2 -2890.313} C_VEL
LIN {X 0,Y 559.546,Z 514.722,A -85,B 0,C 180,E1 -2891.09,E2 -2891.09} C_VEL
LIN {X 0,Y 559.714,Z 502.846,A -85,B 0,C 180,E1 -2891.755,E2 -2891.755} C_VEL
LIN {X 0,Y 559.833,Z 490.579,A -85,B 0,C 180,E1 -2892.272,E2 -2892.272} C_VEL
LIN {X 0,Y 559.879,Z 478.312,A -85,B 0,C 180,E1 -2892.644,E2 -2892.644} C_VEL
LIN {X 0,Y 558.786,Z 471.669,A -85,B 0,C 180,E1 -2892.83,E2 -2892.83} C_VEL
LIN {X 0,Y 558.755,Z 468.455,A -85,B 0,C 180,E1 -2895.316,E2 -2895.316} C_VEL
LIN {X 0,Y 558.774,Z 465.571,A -85,B 0,C 180,E1 -2897.569,E2 -2897.569} C_VEL
LIN {X 0,Y 558.793,Z 462.687,A -85,B 0,C 180,E1 -2899.851,E2 -2899.851} C_VEL
LIN {X 0,Y 558.797,Z 459.976,A -85,B 0,C 180,E1 -2902.167,E2 -2902.167} C_VEL
LIN {X 0,Y 558.865,Z 457.521,A -85,B 0,C 180,E1 -2904.519,E2 -2904.519} C_VEL
LIN {X 0,Y 558.953,Z 455.154,A -85,B 0,C 180,E1 -2906.914,E2 -2906.914} C_VEL
LIN {X 0,Y 558.995,Z 452.133,A -85,B 0,C 180,E1 -2909.829,E2 -2909.829} C_VEL
LIN {X 0,Y 559.037,Z 449.286,A -85,B 0,C 180,E1 -2912.616,E2 -2912.616} C_VEL
LIN {X 0,Y 559.072,Z 446.849,A -85,B 0,C 180,E1 -2915.204,E2 -2915.204} C_VEL
LIN {X 0,Y 559.143,Z 446.84,A -85,B 0,C 180,E1 -2917.64,E2 -2917.64} C_VEL
LIN {X 0,Y 559.165,Z 446.836,A -85,B 0,C 180,E1 -2919.942,E2 -2919.942} C_VEL
LIN {X 0,Y 559.168,Z 446.837,A -85,B 0,C 180,E1 -2922.743,E2 -2922.743} C_VEL
LIN {X 0,Y 559.156,Z 446.836,A -85,B 0,C 180,E1 -2925.761,E2 -2925.761} C_VEL
LIN {X 0,Y 559.169,Z 446.835,A -85,B 0,C 180,E1 -2928.23,E2 -2928.23} C_VEL
LIN {X 0,Y 559.181,Z 446.835,A -85,B 0,C 180,E1 -2931.191,E2 -2931.191} C_VEL
LIN {X 0,Y 559.185,Z 446.863,A -85,B 0,C 180,E1 -2932.148,E2 -2932.148} C_VEL
LIN {X 0,Y 559.922,Z 451.53,A -85,B 0,C 180,E1 -2934.292,E2 -2934.292} C_VEL
LIN {X 0,Y 559.74,Z 457.326,A -85,B 0,C 180,E1 -2936.464,E2 -2936.464} C_VEL
LIN {X 0,Y 559.543,Z 464.85,A -85,B 0,C 180,E1 -2939.004,E2 -2939.004} C_VEL
LIN {X 0,Y 559.434,Z 473.159,A -85,B 0,C 180,E1 -2941.569,E2 -2941.569} C_VEL
LIN {X 0,Y 559.386,Z 481.103,A -85,B 0,C 180,E1 -2943.913,E2 -2943.913} C_VEL
LIN {X 0,Y 559.304,Z 490.368,A -85,B 0,C 180,E1 -2946.534,E2 -2946.534} C_VEL
LIN {X 0,Y 559.227,Z 498.9,A -85,B 0,C 180,E1 -2949.012,E2 -2949.012} C_VEL
LIN {X 0,Y 559.117,Z 508.168,A -85,B 0,C 180,E1 -2951.685,E2 -2951.685} C_VEL
LIN {X 0,Y 559.031,Z 518.759,A -85,B 0,C 180,E1 -2954.692,E2 -2954.692} C_VEL
LIN {X 0,Y 558.955,Z 527.53,A -85,B 0,C 180,E1 -2957.15,E2 -2957.15} C_VEL
LIN {X 0,Y 560.014,Z 535.502,A -85,B 0,C 180,E1 -2957.336,E2 -2957.336} C_VEL
LIN {X 0,Y 559.896,Z 547.872,A -85,B 0,C 180,E1 -2957.679,E2 -2957.679} C_VEL
LIN {X 0,Y 559.76,Z 560.279,A -85,B 0,C 180,E1 -2958.171,E2 -2958.171} C_VEL
LIN {X 0,Y 559.588,Z 572.579,A -85,B 0,C 180,E1 -2958.821,E2 -2958.821} C_VEL
LIN {X 0,Y 559.425,Z 583.922,A -85,B 0,C 180,E1 -2959.596,E2 -2959.596} C_VEL
LIN {X 0,Y 559.244,Z 593.599,A -85,B 0,C 180,E1 -2960.415,E2 -2960.415} C_VEL
LIN {X 0,Y 559.127,Z 602.412,A -85,B 0,C 180,E1 -2961.325,E2 -2961.325} C_VEL
LIN {X 0,Y 558.996,Z 611.001,A -85,B 0,C 180,E1 -2962.414,E2 -2962.414} C_VEL
LIN {X 0,Y 558.884,Z 618.687,A -85,B 0,C 180,E1 -2963.649,E2 -2963.649} C_VEL
LIN {X 0,Y 558.869,Z 623.365,A -85,B 0,C 180,E1 -2964.588,E2 -2964.588} C_VEL
LIN {X 0,Y 558.868,Z 627.677,A -85,B 0,C 180,E1 -2965.673,E2 -2965.673} C_VEL
LIN {X 0,Y 558.836,Z 629.957,A -85,B 0,C 180,E1 -2966.395,E2 -2966.395} C_VEL
LIN {X 0,Y 558.799,Z 631.808,A -85,B 0,C 180,E1 -2967.116,E2 -2967.116} C_VEL
LIN {X 0,Y 558.745,Z 634.185,A -85,B 0,C 180,E1 -2968.558,E2 -2968.558} C_VEL
LIN {X 0,Y 558.74,Z 635,A -85,B 0,C 180,E1 -2970,E2 -2970} C_VEL
LIN {X 0,Y 558.745,Z 634.186,A -85,B 0,C 180,E1 -2971.441,E2 -2971.441} C_VEL
LIN {X 0,Y 558.799,Z 631.81,A -85,B 0,C 180,E1 -2972.884,E2 -2972.884} C_VEL
LIN {X 0,Y 558.843,Z 628.896,A -85,B 0,C 180,E1 -2973.966,E2 -2973.966} C_VEL
LIN {X 0,Y 558.799,Z 624.949,A -85,B 0,C 180,E1 -2975.051,E2 -2975.051} C_VEL
LIN {X 0,Y 558.921,Z 619.867,A -85,B 0,C 180,E1 -2976.135,E2 -2976.135} C_VEL
LIN {X 0,Y 558.977,Z 613.469,A -85,B 0,C 180,E1 -2977.223,E2 -2977.223} C_VEL
LIN {X 0,Y 559.099,Z 605.478,A -85,B 0,C 180,E1 -2978.312,E2 -2978.312} C_VEL
LIN {X 0,Y 559.195,Z 597.336,A -85,B 0,C 180,E1 -2979.221,E2 -2979.221} C_VEL
LIN {X 0,Y 559.351,Z 587.401,A -85,B 0,C 180,E1 -2980.131,E2 -2980.131} C_VEL
LIN {X 0,Y 559.537,Z 576.402,A -85,B 0,C 180,E1 -2980.937,E2 -2980.937} C_VEL
LIN {X 0,Y 559.671,Z 564.463,A -85,B 0,C 180,E1 -2981.628,E2 -2981.628} C_VEL
LIN {X 0,Y 559.825,Z 551.768,A -85,B 0,C 180,E1 -2982.184,E2 -2982.184} C_VEL
LIN {X 0,Y 559.973,Z 538.349,A -85,B 0,C 180,E1 -2982.595,E2 -2982.595} C_VEL
LIN {X 0,Y 559.749,Z 532.511,A -85,B 0,C 180,E1 -2982.73,E2 -2982.73} C_VEL
LIN {X 0,Y 558.955,Z 527.53,A -85,B 0,C 180,E1 -2982.85,E2 -2982.85} C_VEL
LIN {X 0,Y 559.055,Z 517.436,A -85,B 0,C 180,E1 -2985.681,E2 -2985.681} C_VEL
LIN {X 0,Y 559.134,Z 506.844,A -85,B 0,C 180,E1 -2988.694,E2 -2988.694} C_VEL
LIN {X 0,Y 559.226,Z 496.916,A -85,B 0,C 180,E1 -2991.567,E2 -2991.567} C_VEL
LIN {X 0,Y 559.369,Z 486.924,A -85,B 0,C 180,E1 -2994.495,E2 -2994.495} C_VEL
LIN {X 0,Y 559.522,Z 476.198,A -85,B 0,C 180,E1 -2997.694,E2 -2997.694} C_VEL
LIN {X 0,Y 559.65,Z 466.799,A -85,B 0,C 180,E1 -3000.57,E2 -3000.57} C_VEL
LIN {X 0,Y 559.844,Z 457.645,A -85,B 0,C 180,E1 -3003.529,E2 -3003.529} C_VEL
LIN {X 0,Y 559.858,Z 451.135,A -85,B 0,C 180,E1 -3005.712,E2 -3005.712} C_VEL
LIN {X 0,Y 559.178,Z 446.834,A -85,B 0,C 180,E1 -3007.301,E2 -3007.301} C_VEL
LIN {X 0,Y 559.172,Z 446.836,A -85,B 0,C 180,E1 -3009.943,E2 -3009.943} C_VEL
LIN {X 0,Y 559.16,Z 446.836,A -85,B 0,C 180,E1 -3012.744,E2 -3012.744} C_VEL
LIN {X 0,Y 559.158,Z 446.835,A -85,B 0,C 180,E1 -3015.76,E2 -3015.76} C_VEL
LIN {X 0,Y 559.192,Z 446.829,A -85,B 0,C 180,E1 -3018.232,E2 -3018.232} C_VEL
LIN {X 0,Y 559.175,Z 446.831,A -85,B 0,C 180,E1 -3021.192,E2 -3021.192} C_VEL
LIN {X 0,Y 559.143,Z 446.839,A -85,B 0,C 180,E1 -3023.789,E2 -3023.789} C_VEL
LIN {X 0,Y 559.165,Z 446.832,A -85,B 0,C 180,E1 -3026.425,E2 -3026.425} C_VEL
LIN {X 0,Y 559.158,Z 446.834,A -85,B 0,C 180,E1 -3028.981,E2 -3028.981} C_VEL
LIN {X 0,Y 559.17,Z 446.836,A -85,B 0,C 180,E1 -3031.619,E2 -3031.619} C_VEL
LIN {X 0,Y 559.183,Z 446.829,A -85,B 0,C 180,E1 -3033.903,E2 -3033.903} C_VEL
LIN {X 0,Y 559.144,Z 446.838,A -85,B 0,C 180,E1 -3036.571,E2 -3036.571} C_VEL
LIN {X 0,Y 559.183,Z 446.835,A -85,B 0,C 180,E1 -3039.396,E2 -3039.396} C_VEL
LIN {X 0,Y 559.148,Z 446.833,A -85,B 0,C 180,E1 -3041.686,E2 -3041.686} C_VEL
LIN {X 0,Y 559.17,Z 446.834,A -85,B 0,C 180,E1 -3043.948,E2 -3043.948} C_VEL
LIN {X 0,Y 559.176,Z 446.832,A -85,B 0,C 180,E1 -3046.184,E2 -3046.184} C_VEL
LIN {X 0,Y 559.197,Z 446.829,A -85,B 0,C 180,E1 -3049.134,E2 -3049.134} C_VEL
LIN {X 0,Y 559.207,Z 446.832,A -85,B 0,C 180,E1 -3052.054,E2 -3052.054} C_VEL
LIN {X 0,Y 559.257,Z 446.825,A -85,B 0,C 180,E1 -3054.953,E2 -3054.953} C_VEL
LIN {X 0,Y 559.252,Z 446.822,A -85,B 0,C 180,E1 -3057.84,E2 -3057.84} C_VEL
LIN {X 0,Y 559.277,Z 446.818,A -85,B 0,C 180,E1 -3060.72,E2 -3060.72} C_VEL
LIN {X 0,Y 559.244,Z 446.827,A -85,B 0,C 180,E1 -3062.881,E2 -3062.881} C_VEL
LIN {X 0,Y 559.23,Z 446.826,A -85,B 0,C 180,E1 -3065.77,E2 -3065.77} C_VEL
LIN {X 0,Y 559.194,Z 446.829,A -85,B 0,C 180,E1 -3068.674,E2 -3068.674} C_VEL
LIN {X 0,Y 559.208,Z 446.826,A -85,B 0,C 180,E1 -3071.601,E2 -3071.601} C_VEL
LIN {X 0,Y 559.203,Z 446.827,A -85,B 0,C 180,E1 -3074.596,E2 -3074.596} C_VEL
LIN {X 0,Y 559.162,Z 446.832,A -85,B 0,C 180,E1 -3077.557,E2 -3077.557} C_VEL
LIN {X 0,Y 559.176,Z 446.833,A -85,B 0,C 180,E1 -3079.837,E2 -3079.837} C_VEL
LIN {X 0,Y 559.145,Z 446.835,A -85,B 0,C 180,E1 -3082.153,E2 -3082.153} C_VEL
LIN {X 0,Y 559.179,Z 446.83,A -85,B 0,C 180,E1 -3085.298,E2 -3085.298} C_VEL
LIN {X 0,Y 559.192,Z 446.832,A -85,B 0,C 180,E1 -3087.712,E2 -3087.712} C_VEL
LIN {X 0,Y 559.143,Z 446.835,A -85,B 0,C 180,E1 -3090.618,E2 -3090.618} C_VEL
LIN {X 0,Y 558.483,Z 446.921,A -85,B 0,C 180,E1 -3091.22,E2 -3091.22} C_VEL
LIN {X 0,Y 555.624,Z 447.275,A -85,B 0,C 180,E1 -3092.196,E2 -3092.196} C_VEL
LIN {X 0,Y 553.213,Z 447.573,A -85,B 0,C 180,E1 -3092.982,E2 -3092.982} C_VEL
LIN {X 0,Y 552.192,Z 447.7,A -85,B 0,C 180,E1 -3093.588,E2 -3093.588} C_VEL
LIN {X 0,Y 552.116,Z 447.711,A -85,B 0,C 180,E1 -3093.794,E2 -3093.794} C_VEL
LIN {X 0,Y 552.115,Z 447.711,A -85,B 0,C 180,E1 -3096.747,E2 -3096.747} C_VEL
LIN {X 0,Y 552.133,Z 447.707,A -85,B 0,C 180,E1 -3099.527,E2 -3099.527} C_VEL
LIN {X 0,Y 552.135,Z 447.708,A -85,B 0,C 180,E1 -3102.425,E2 -3102.425} C_VEL
LIN {X 0,Y 552.102,Z 447.712,A -85,B 0,C 180,E1 -3105.563,E2 -3105.563} C_VEL
LIN {X 0,Y 552.124,Z 447.71,A -85,B 0,C 180,E1 -3108.554,E2 -3108.554} C_VEL
LIN {X 0,Y 552.121,Z 447.713,A -85,B 0,C 180,E1 -3111.411,E2 -3111.411} C_VEL
LIN {X 0,Y 552.104,Z 447.714,A -85,B 0,C 180,E1 -3114.158,E2 -3114.158} C_VEL
LIN {X 0,Y 552.12,Z 447.709,A -85,B 0,C 180,E1 -3116.814,E2 -3116.814} C_VEL
LIN {X 0,Y 552.106,Z 447.713,A -85,B 0,C 180,E1 -3119.391,E2 -3119.391} C_VEL
LIN {X 0,Y 552.107,Z 447.713,A -85,B 0,C 180,E1 -3121.902,E2 -3121.902} C_VEL
LIN {X 0,Y 552.161,Z 447.704,A -85,B 0,C 180,E1 -3124.65,E2 -3124.65} C_VEL
LIN {X 0,Y 552.097,Z 447.712,A -85,B 0,C 180,E1 -3127.549,E2 -3127.549} C_VEL
LIN {X 0,Y 552.149,Z 447.707,A -85,B 0,C 180,E1 -3130.375,E2 -3130.375} C_VEL
LIN {X 0,Y 552.16,Z 447.709,A -85,B 0,C 180,E1 -3132.977,E2 -3132.977} C_VEL
LIN {X 0,Y 552.141,Z 447.71,A -85,B 0,C 180,E1 -3136.005,E2 -3136.005} C_VEL
LIN {X 0,Y 552.168,Z 447.705,A -85,B 0,C 180,E1 -3138.994,E2 -3138.994} C_VEL
LIN {X 0,Y 552.163,Z 447.705,A -85,B 0,C 180,E1 -3141.952,E2 -3141.952} C_VEL
LIN {X 0,Y 552.229,Z 447.695,A -85,B 0,C 180,E1 -3144.889,E2 -3144.889} C_VEL
LIN {X 0,Y 552.23,Z 447.696,A -85,B 0,C 180,E1 -3147.812,E2 -3147.812} C_VEL
LIN {X 0,Y 552.245,Z 447.694,A -85,B 0,C 180,E1 -3150.729,E2 -3150.729} C_VEL
LIN {X 0,Y 552.207,Z 447.699,A -85,B 0,C 180,E1 -3152.918,E2 -3152.918} C_VEL
LIN {X 0,Y 552.204,Z 447.699,A -85,B 0,C 180,E1 -3155.844,E2 -3155.844} C_VEL
LIN {X 0,Y 552.151,Z 447.705,A -85,B 0,C 180,E1 -3158.786,E2 -3158.786} C_VEL
LIN {X 0,Y 552.169,Z 447.704,A -85,B 0,C 180,E1 -3161.75,E2 -3161.75} C_VEL
LIN {X 0,Y 552.142,Z 447.707,A -85,B 0,C 180,E1 -3164.748,E2 -3164.748} C_VEL
LIN {X 0,Y 552.114,Z 447.712,A -85,B 0,C 180,E1 -3167.789,E2 -3167.789} C_VEL
LIN {X 0,Y 552.133,Z 447.709,A -85,B 0,C 180,E1 -3170.101,E2 -3170.101} C_VEL
LIN {X 0,Y 552.098,Z 447.713,A -85,B 0,C 180,E1 -3172.451,E2 -3172.451} C_VEL
LIN {X 0,Y 552.161,Z 447.708,A -85,B 0,C 180,E1 -3175.35,E2 -3175.35} C_VEL
LIN {X 0,Y 552.115,Z 447.713,A -85,B 0,C 180,E1 -3178.098,E2 -3178.098} C_VEL
LIN {X 0,Y 552.108,Z 447.71,A -85,B 0,C 180,E1 -3180.609,E2 -3180.609} C_VEL
LIN {X 0,Y 552.12,Z 447.713,A -85,B 0,C 180,E1 -3183.186,E2 -3183.186} C_VEL
LIN {X 0,Y 552.091,Z 447.715,A -85,B 0,C 180,E1 -3185.844,E2 -3185.844} C_VEL
LIN {X 0,Y 552.129,Z 447.712,A -85,B 0,C 180,E1 -3189.062,E2 -3189.062} C_VEL
LIN {X 0,Y 552.135,Z 447.708,A -85,B 0,C 180,E1 -3191.445,E2 -3191.445} C_VEL
LIN {X 0,Y 552.096,Z 447.712,A -85,B 0,C 180,E1 -3194.531,E2 -3194.531} C_VEL
LIN {X 0,Y 552.136,Z 447.708,A -85,B 0,C 180,E1 -3197.584,E2 -3197.584} C_VEL
LIN {X 0,Y 552.133,Z 447.709,A -85,B 0,C 180,E1 -3200.473,E2 -3200.473} C_VEL
LIN {X 0,Y 552.107,Z 447.716,A -85,B 0,C 180,E1 -3203.317,E2 -3203.317} C_VEL
LIN {X 0,Y 551.963,Z 447.733,A -85,B 0,C 180,E1 -3205.927,E2 -3205.927} C_VEL
LIN {X 0,Y 551.838,Z 447.789,A -85,B 0,C 180,E1 -3206.795,E2 -3206.795} C_VEL
LIN {X 0,Y 551.833,Z 450.683,A -85,B 0,C 180,E1 -3209.374,E2 -3209.374} C_VEL
LIN {X 0,Y 551.821,Z 453.52,A -85,B 0,C 180,E1 -3211.885,E2 -3211.885} C_VEL
LIN {X 0,Y 551.78,Z 456.748,A -85,B 0,C 180,E1 -3214.733,E2 -3214.733} C_VEL
LIN {X 0,Y 551.728,Z 459.94,A -85,B 0,C 180,E1 -3217.533,E2 -3217.533} C_VEL
LIN {X 0,Y 551.732,Z 463.535,A -85,B 0,C 180,E1 -3220.659,E2 -3220.659} C_VEL
LIN {X 0,Y 551.709,Z 467.378,A -85,B 0,C 180,E1 -3223.725,E2 -3223.725} C_VEL
LIN {X 0,Y 551.7,Z 470.261,A -85,B 0,C 180,E1 -3225.993,E2 -3225.993} C_VEL
LIN {X 0,Y 551.709,Z 471.672,A -85,B 0,C 180,E1 -3227.095,E2 -3227.095} C_VEL
LIN {X 0,Y 553.029,Z 480.231,A -85,B 0,C 180,E1 -3227.337,E2 -3227.337} C_VEL
LIN {X 0,Y 552.902,Z 493.009,A -85,B 0,C 180,E1 -3227.753,E2 -3227.753} C_VEL
LIN {X 0,Y 552.701,Z 505.654,A -85,B 0,C 180,E1 -3228.331,E2 -3228.331} C_VEL
LIN {X 0,Y 552.539,Z 516.903,A -85,B 0,C 180,E1 -3229.001,E2 -3229.001} C_VEL
LIN {X 0,Y 552.306,Z 527.947,A -85,B 0,C 180,E1 -3229.831,E2 -3229.831} C_VEL
LIN {X 0,Y 552.153,Z 538.679,A -85,B 0,C 180,E1 -3230.845,E2 -3230.845} C_VEL
LIN {X 0,Y 552.007,Z 546.599,A -85,B 0,C 180,E1 -3231.765,E2 -3231.765} C_VEL
LIN {X 0,Y 551.895,Z 554.458,A -85,B 0,C 180,E1 -3232.886,E2 -3232.886} C_VEL
LIN {X 0,Y 551.868,Z 561.456,A -85,B 0,C 180,E1 -3234.152,E2 -3234.152} C_VEL
LIN {X 0,Y 551.725,Z 566.197,A -85,B 0,C 180,E1 -3235.25,E2 -3235.25} C_VEL
LIN {X 0,Y 551.751,Z 569.829,A -85,B 0,C 180,E1 -3236.348,E2 -3236.348} C_VEL
LIN {X 0,Y 551.724,Z 571.705,A -85,B 0,C 180,E1 -3237.079,E2 -3237.079} C_VEL
LIN {X 0,Y 551.656,Z 573.129,A -85,B 0,C 180,E1 -3237.81,E2 -3237.81} C_VEL
LIN {X 0,Y 551.643,Z 574.757,A -85,B 0,C 180,E1 -3239.27,E2 -3239.27} C_VEL
LIN {X 0,Y 551.641,Z 574.996,A -85,B 0,C 180,E1 -3240,E2 -3240} C_VEL
LIN {X 0,Y 551.641,Z 574.814,A -85,B 0,C 180,E1 -3240.73,E2 -3240.73} C_VEL
LIN {X 0,Y 551.655,Z 573.266,A -85,B 0,C 180,E1 -3242.19,E2 -3242.19} C_VEL
LIN {X 0,Y 551.724,Z 571.904,A -85,B 0,C 180,E1 -3242.921,E2 -3242.921} C_VEL
LIN {X 0,Y 551.764,Z 569.026,A -85,B 0,C 180,E1 -3244.017,E2 -3244.017} C_VEL
LIN {X 0,Y 551.723,Z 565.125,A -85,B 0,C 180,E1 -3245.116,E2 -3245.116} C_VEL
LIN {X 0,Y 551.812,Z 559.387,A -85,B 0,C 180,E1 -3246.35,E2 -3246.35} C_VEL
LIN {X 0,Y 551.925,Z 552.538,A -85,B 0,C 180,E1 -3247.5,E2 -3247.5} C_VEL
LIN {X 0,Y 552.063,Z 544.355,A -85,B 0,C 180,E1 -3248.603,E2 -3248.603} C_VEL
LIN {X 0,Y 552.196,Z 535.987,A -85,B 0,C 180,E1 -3249.524,E2 -3249.524} C_VEL
LIN {X 0,Y 552.401,Z 525.666,A -85,B 0,C 180,E1 -3250.445,E2 -3250.445} C_VEL
LIN {X 0,Y 552.611,Z 513.899,A -85,B 0,C 180,E1 -3251.284,E2 -3251.284} C_VEL
LIN {X 0,Y 552.756,Z 502.445,A -85,B 0,C 180,E1 -3251.924,E2 -3251.924} C_VEL
LIN {X 0,Y 552.916,Z 490.432,A -85,B 0,C 180,E1 -3252.432,E2 -3252.432} C_VEL
LIN {X 0,Y 552.91,Z 478.746,A -85,B 0,C 180,E1 -3252.794,E2 -3252.794} C_VEL
LIN {X 0,Y 551.695,Z 471.668,A -85,B 0,C 180,E1 -3252.998,E2 -3252.998} C_VEL
LIN {X 0,Y 551.671,Z 468.454,A -85,B 0,C 180,E1 -3255.517,E2 -3255.517} C_VEL
LIN {X 0,Y 551.684,Z 465.57,A -85,B 0,C 180,E1 -3257.803,E2 -3257.803} C_VEL
LIN {X 0,Y 551.724,Z 462.829,A -85,B 0,C 180,E1 -3260.117,E2 -3260.117} C_VEL
LIN {X 0,Y 551.732,Z 460.408,A -85,B 0,C 180,E1 -3262.466,E2 -3262.466} C_VEL
LIN {X 0,Y 551.841,Z 457.497,A -85,B 0,C 180,E1 -3265.28,E2 -3265.28} C_VEL
LIN {X 0,Y 551.892,Z 454.639,A -85,B 0,C 180,E1 -3268.11,E2 -3268.11} C_VEL
LIN {X 0,Y 551.946,Z 452.168,A -85,B 0,C 180,E1 -3270.619,E2 -3270.619} C_VEL
LIN {X 0,Y 551.998,Z 449.586,A -85,B 0,C 180,E1 -3273.194,E2 -3273.194} C_VEL
LIN {X 0,Y 552.024,Z 447.881,A -85,B 0,C 180,E1 -3274.953,E2 -3274.953} C_VEL
LIN {X 0,Y 552.097,Z 447.717,A -85,B 0,C 180,E1 -3277.664,E2 -3277.664} C_VEL
LIN {X 0,Y 552.114,Z 447.714,A -85,B 0,C 180,E1 -3280.481,E2 -3280.481} C_VEL
LIN {X 0,Y 552.118,Z 447.713,A -85,B 0,C 180,E1 -3283.484,E2 -3283.484} C_VEL
LIN {X 0,Y 552.109,Z 447.715,A -85,B 0,C 180,E1 -3286.576,E2 -3286.576} C_VEL
LIN {X 0,Y 552.124,Z 447.713,A -85,B 0,C 180,E1 -3289.52,E2 -3289.52} C_VEL
LIN {X 0,Y 552.137,Z 447.802,A -85,B 0,C 180,E1 -3291.793,E2 -3291.793} C_VEL
LIN {X 0,Y 552.855,Z 451.81,A -85,B 0,C 180,E1 -3293.763,E2 -3293.763} C_VEL
LIN {X 0,Y 552.941,Z 455.062,A -85,B 0,C 180,E1 -3295.113,E2 -3295.113} C_VEL
LIN {X 0,Y 552.661,Z 462.208,A -85,B 0,C 180,E1 -3297.717,E2 -3297.717} C_VEL
LIN {X 0,Y 552.479,Z 469.922,A -85,B 0,C 180,E1 -3300.257,E2 -3300.257} C_VEL
LIN {X 0,Y 552.373,Z 479.711,A -85,B 0,C 180,E1 -3303.252,E2 -3303.252} C_VEL
LIN {X 0,Y 552.277,Z 489.125,A -85,B 0,C 180,E1 -3305.97,E2 -3305.97} C_VEL
LIN {X 0,Y 552.199,Z 498.888,A -85,B 0,C 180,E1 -3308.732,E2 -3308.732} C_VEL
LIN {X 0,Y 552.086,Z 508.168,A -85,B 0,C 180,E1 -3311.443,E2 -3311.443} C_VEL
LIN {X 0,Y 551.982,Z 518.759,A -85,B 0,C 180,E1 -3314.492,E2 -3314.492} C_VEL
LIN {X 0,Y 551.909,Z 527.53,A -85,B 0,C 180,E1 -3316.983,E2 -3316.983} C_VEL
LIN {X 0,Y 553.097,Z 535.502,A -85,B 0,C 180,E1 -3317.175,E2 -3317.175} C_VEL
LIN {X 0,Y 552.972,Z 547.871,A -85,B 0,C 180,E1 -3317.522,E2 -3317.522} C_VEL
LIN {X 0,Y 552.813,Z 559.503,A -85,B 0,C 180,E1 -3317.984,E2 -3317.984} C_VEL
LIN {X 0,Y 552.633,Z 571.894,A -85,B 0,C 180,E1 -3318.638,E2 -3318.638} C_VEL
LIN {X 0,Y 552.415,Z 582.744,A -85,B 0,C 180,E1 -3319.369,E2 -3319.369} C_VEL
LIN {X 0,Y 552.233,Z 593.599,A -85,B 0,C 180,E1 -3320.292,E2 -3320.292} C_VEL
LIN {X 0,Y 552.079,Z 602.412,A -85,B 0,C 180,E1 -3321.213,E2 -3321.213} C_VEL
LIN {X 0,Y 551.949,Z 611.001,A -85,B 0,C 180,E1 -3322.317,E2 -3322.317} C_VEL
LIN {X 0,Y 551.823,Z 617.868,A -85,B 0,C 180,E1 -3323.418,E2 -3323.418} C_VEL
LIN {X 0,Y 551.804,Z 623.365,A -85,B 0,C 180,E1 -3324.518,E2 -3324.518} C_VEL
LIN {X 0,Y 551.764,Z 627.677,A -85,B 0,C 180,E1 -3325.617,E2 -3325.617} C_VEL
LIN {X 0,Y 551.75,Z 629.957,A -85,B 0,C 180,E1 -3326.348,E2 -3326.348} C_VEL
LIN {X 0,Y 551.723,Z 631.807,A -85,B 0,C 180,E1 -3327.079,E2 -3327.079} C_VEL
LIN {X 0,Y 551.645,Z 634.184,A -85,B 0,C 180,E1 -3328.54,E2 -3328.54} C_VEL
LIN {X 0,Y 551.64,Z 635,A -85,B 0,C 180,E1 -3330,E2 -3330} C_VEL
LIN {X 0,Y 551.645,Z 634.186,A -85,B 0,C 180,E1 -3331.46,E2 -3331.46} C_VEL
LIN {X 0,Y 551.723,Z 631.81,A -85,B 0,C 180,E1 -3332.921,E2 -3332.921} C_VEL
LIN {X 0,Y 551.763,Z 628.896,A -85,B 0,C 180,E1 -3334.017,E2 -3334.017} C_VEL
LIN {X 0,Y 551.724,Z 624.949,A -85,B 0,C 180,E1 -3335.116,E2 -3335.116} C_VEL
LIN {X 0,Y 551.803,Z 619.189,A -85,B 0,C 180,E1 -3336.342,E2 -3336.342} C_VEL
LIN {X 0,Y 551.926,Z 612.237,A -85,B 0,C 180,E1 -3337.5,E2 -3337.5} C_VEL
LIN {X 0,Y 552.082,Z 603.991,A -85,B 0,C 180,E1 -3338.602,E2 -3338.602} C_VEL
LIN {X 0,Y 552.201,Z 595.539,A -85,B 0,C 180,E1 -3339.524,E2 -3339.524} C_VEL
LIN {X 0,Y 552.419,Z 585.096,A -85,B 0,C 180,E1 -3340.445,E2 -3340.445} C_VEL
LIN {X 0,Y 552.59,Z 574.298,A -85,B 0,C 180,E1 -3341.213,E2 -3341.213} C_VEL
LIN {X 0,Y 552.753,Z 563.409,A -85,B 0,C 180,E1 -3341.831,E2 -3341.831} C_VEL
LIN {X 0,Y 552.903,Z 551.765,A -85,B 0,C 180,E1 -3342.34,E2 -3342.34} C_VEL
LIN {X 0,Y 553.057,Z 538.348,A -85,B 0,C 180,E1 -3342.756,E2 -3342.756} C_VEL
LIN {X 0,Y 552.905,Z 533.796,A -85,B 0,C 180,E1 -3342.864,E2 -3342.864} C_VEL
LIN {X 0,Y 551.909,Z 527.53,A -85,B 0,C 180,E1 -3343.017,E2 -3343.017} C_VEL
LIN {X 0,Y 551.995,Z 517.436,A -85,B 0,C 180,E1 -3345.887,E2 -3345.887} C_VEL
LIN {X 0,Y 552.085,Z 506.844,A -85,B 0,C 180,E1 -3348.942,E2 -3348.942} C_VEL
LIN {X 0,Y 552.188,Z 497.368,A -85,B 0,C 180,E1 -3351.703,E2 -3351.703} C_VEL
LIN {X 0,Y 552.327,Z 488.103,A -85,B 0,C 180,E1 -3354.427,E2 -3354.427} C_VEL
LIN {X 0,Y 552.493,Z 478.778,A -85,B 0,C 180,E1 -3357.254,E2 -3357.254} C_VEL
LIN {X 0,Y 552.678,Z 468.09,A -85,B 0,C 180,E1 -3360.574,E2 -3360.574} C_VEL
LIN {X 0,Y 552.895,Z 458.917,A -85,B 0,C 180,E1 -3363.569,E2 -3363.569} C_VEL
LIN {X 0,Y 552.881,Z 452.413,A -85,B 0,C 180,E1 -3365.784,E2 -3365.784} C_VEL
LIN {X 0,Y 552.115,Z 447.714,A -85,B 0,C 180,E1 -3367.547,E2 -3367.547} C_VEL
LIN {X 0,Y 552.123,Z 447.71,A -85,B 0,C 180,E1 -3370.48,E2 -3370.48} C_VEL
LIN {X 0,Y 552.121,Z 447.71,A -85,B 0,C 180,E1 -3373.485,E2 -3373.485} C_VEL
LIN {X 0,Y 552.123,Z 447.71,A -85,B 0,C 180,E1 -3376.578,E2 -3376.578} C_VEL
LIN {X 0,Y 552.112,Z 447.712,A -85,B 0,C 180,E1 -3379.519,E2 -3379.519} C_VEL
LIN {X 0,Y 552.094,Z 447.717,A -85,B 0,C 180,E1 -3382.336,E2 -3382.336} C_VEL
LIN {X 0,Y 552.087,Z 447.715,A -85,B 0,C 180,E1 -3385.051,E2 -3385.051} C_VEL
LIN {X 0,Y 552.118,Z 447.709,A -85,B 0,C 180,E1 -3387.681,E2 -3387.681} C_VEL
LIN {X 0,Y 552.114,Z 447.715,A -85,B 0,C 180,E1 -3390.235,E2 -3390.235} C_VEL
LIN {X 0,Y 552.142,Z 447.71,A -85,B 0,C 180,E1 -3393,E2 -3393} C_VEL
LIN {X 0,Y 552.116,Z 447.711,A -85,B 0,C 180,E1 -3395.161,E2 -3395.161} C_VEL
LIN {X 0,Y 552.128,Z 447.71,A -85,B 0,C 180,E1 -3398.337,E2 -3398.337} C_VEL
LIN {X 0,Y 552.159,Z 447.706,A -85,B 0,C 180,E1 -3400.675,E2 -3400.675} C_VEL
LIN {X 0,Y 552.119,Z 447.71,A -85,B 0,C 180,E1 -3403.737,E2 -3403.737} C_VEL
LIN {X 0,Y 552.139,Z 447.71,A -85,B 0,C 180,E1 -3406.005,E2 -3406.005} C_VEL
LIN {X 0,Y 552.165,Z 447.707,A -85,B 0,C 180,E1 -3408.994,E2 -3408.994} C_VEL
LIN {X 0,Y 552.161,Z 447.709,A -85,B 0,C 180,E1 -3411.952,E2 -3411.952} C_VEL
LIN {X 0,Y 552.232,Z 447.699,A -85,B 0,C 180,E1 -3414.889,E2 -3414.889} C_VEL
LIN {X 0,Y 552.224,Z 447.697,A -85,B 0,C 180,E1 -3417.812,E2 -3417.812} C_VEL
LIN {X 0,Y 552.247,Z 447.694,A -85,B 0,C 180,E1 -3420.729,E2 -3420.729} C_VEL
LIN {X 0,Y 552.21,Z 447.703,A -85,B 0,C 180,E1 -3422.918,E2 -3422.918} C_VEL
LIN {X 0,Y 552.2,Z 447.703,A -85,B 0,C 180,E1 -3425.844,E2 -3425.844} C_VEL
LIN {X 0,Y 552.164,Z 447.706,A -85,B 0,C 180,E1 -3428.786,E2 -3428.786} C_VEL
LIN {X 0,Y 552.166,Z 447.703,A -85,B 0,C 180,E1 -3431.751,E2 -3431.751} C_VEL
LIN {X 0,Y 552.14,Z 447.707,A -85,B 0,C 180,E1 -3434.749,E2 -3434.749} C_VEL
LIN {X 0,Y 552.113,Z 447.71,A -85,B 0,C 180,E1 -3437.789,E2 -3437.789} C_VEL
LIN {X 0,Y 552.134,Z 447.713,A -85,B 0,C 180,E1 -3440.101,E2 -3440.101} C_VEL
LIN {X 0,Y 552.096,Z 447.712,A -85,B 0,C 180,E1 -3442.451,E2 -3442.451} C_VEL
LIN {X 0,Y 552.159,Z 447.704,A -85,B 0,C 180,E1 -3445.351,E2 -3445.351} C_VEL
LIN {X 0,Y 552.127,Z 447.711,A -85,B 0,C 180,E1 -3448.098,E2 -3448.098} C_VEL
LIN {X 0,Y 552.106,Z 447.713,A -85,B 0,C 180,E1 -3450.614,E2 -3450.614} C_VEL
LIN {X 0,Y 552.126,Z 447.708,A -85,B 0,C 180,E1 -3453.185,E2 -3453.185} C_VEL
LIN {X 0,Y 552.116,Z 447.711,A -85,B 0,C 180,E1 -3453.794,E2 -3453.794} C_VEL
LIN {X 0,Y 551.48,Z 447.795,A -85,B 0,C 180,E1 -3454.402,E2 -3454.402} C_VEL
LIN {X 0,Y 548.659,Z 448.147,A -85,B 0,C 180,E1 -3455.39,E2 -3455.39} C_VEL
LIN {X 0,Y 546.24,Z 448.446,A -85,B 0,C 180,E1 -3456.186,E2 -3456.186} C_VEL
LIN {X 0,Y 545.171,Z 448.578,A -85,B 0,C 180,E1 -3456.8,E2 -3456.8} C_VEL
LIN {X 0,Y 545.069,Z 448.59,A -85,B 0,C 180,E1 -3457.008,E2 -3457.008} C_VEL
LIN {X 0,Y 545.069,Z 448.591,A -85,B 0,C 180,E1 -3460.143,E2 -3460.143} C_VEL
LIN {X 0,Y 545.091,Z 448.587,A -85,B 0,C 180,E1 -3463.106,E2 -3463.106} C_VEL
LIN {X 0,Y 545.071,Z 448.589,A -85,B 0,C 180,E1 -3466.224,E2 -3466.224} C_VEL
LIN {X 0,Y 545.085,Z 448.585,A -85,B 0,C 180,E1 -3468.886,E2 -3468.886} C_VEL
LIN {X 0,Y 545.084,Z 448.587,A -85,B 0,C 180,E1 -3470.819,E2 -3470.819} C_VEL
LIN {X 0,Y 545.053,Z 448.589,A -85,B 0,C 180,E1 -3473.62,E2 -3473.62} C_VEL
LIN {X 0,Y 545.072,Z 448.589,A -85,B 0,C 180,E1 -3476.329,E2 -3476.329} C_VEL
LIN {X 0,Y 545.07,Z 448.592,A -85,B 0,C 180,E1 -3478.952,E2 -3478.952} C_VEL
LIN {X 0,Y 545.105,Z 448.583,A -85,B 0,C 180,E1 -3481.508,E2 -3481.508} C_VEL
LIN {X 0,Y 545.1,Z 448.584,A -85,B 0,C 180,E1 -3484.491,E2 -3484.491} C_VEL
LIN {X 0,Y 545.043,Z 448.592,A -85,B 0,C 180,E1 -3487.242,E2 -3487.242} C_VEL
LIN {X 0,Y 545.121,Z 448.582,A -85,B 0,C 180,E1 -3490.415,E2 -3490.415} C_VEL
LIN {X 0,Y 545.075,Z 448.588,A -85,B 0,C 180,E1 -3493.521,E2 -3493.521} C_VEL
LIN {X 0,Y 545.1,Z 448.585,A -85,B 0,C 180,E1 -3495.82,E2 -3495.82} C_VEL
LIN {X 0,Y 545.124,Z 448.582,A -85,B 0,C 180,E1 -3498.85,E2 -3498.85} C_VEL
LIN {X 0,Y 545.133,Z 448.58,A -85,B 0,C 180,E1 -3501.847,E2 -3501.847} C_VEL
LIN {X 0,Y 545.205,Z 448.57,A -85,B 0,C 180,E1 -3504.823,E2 -3504.823} C_VEL
LIN {X 0,Y 545.202,Z 448.572,A -85,B 0,C 180,E1 -3507.784,E2 -3507.784} C_VEL
LIN {X 0,Y 545.216,Z 448.569,A -85,B 0,C 180,E1 -3510.739,E2 -3510.739} C_VEL
LIN {X 0,Y 545.174,Z 448.576,A -85,B 0,C 180,E1 -3512.956,E2 -3512.956} C_VEL
LIN {X 0,Y 545.176,Z 448.575,A -85,B 0,C 180,E1 -3515.92,E2 -3515.92} C_VEL
LIN {X 0,Y 545.113,Z 448.581,A -85,B 0,C 180,E1 -3518.9,E2 -3518.9} C_VEL
LIN {X 0,Y 545.141,Z 448.579,A -85,B 0,C 180,E1 -3521.904,E2 -3521.904} C_VEL
LIN {X 0,Y 545.091,Z 448.584,A -85,B 0,C 180,E1 -3524.944,E2 -3524.944} C_VEL
LIN {X 0,Y 545.082,Z 448.586,A -85,B 0,C 180,E1 -3528.026,E2 -3528.026} C_VEL
LIN {X 0,Y 545.098,Z 448.588,A -85,B 0,C 180,E1 -3530.372,E2 -3530.372} C_VEL
LIN {X 0,Y 545.087,Z 448.589,A -85,B 0,C 180,E1 -3533.559,E2 -3533.559} C_VEL
LIN {X 0,Y 545.085,Z 448.586,A -85,B 0,C 180,E1 -3536,E2 -3536} C_VEL
LIN {X 0,Y 545.095,Z 448.585,A -85,B 0,C 180,E1 -3538.748,E2 -3538.748} C_VEL
LIN {X 0,Y 545.063,Z 448.591,A -85,B 0,C 180,E1 -3541.679,E2 -3541.679} C_VEL
LIN {X 0,Y 545.068,Z 448.592,A -85,B 0,C 180,E1 -3544.564,E2 -3544.564} C_VEL
LIN {X 0,Y 545.041,Z 448.592,A -85,B 0,C 180,E1 -3547.304,E2 -3547.304} C_VEL
LIN {X 0,Y 545.073,Z 448.587,A -85,B 0,C 180,E1 -3550.142,E2 -3550.142} C_VEL
LIN {X 0,Y 545.083,Z 448.586,A -85,B 0,C 180,E1 -3553.106,E2 -3553.106} C_VEL
LIN {X 0,Y 545.072,Z 448.587,A -85,B 0,C 180,E1 -3556.224,E2 -3556.224} C_VEL
LIN {X 0,Y 545.092,Z 448.587,A -85,B 0,C 180,E1 -3558.886,E2 -3558.886} C_VEL
LIN {X 0,Y 545.055,Z 448.594,A -85,B 0,C 180,E1 -3561.763,E2 -3561.763} C_VEL
LIN {X 0,Y 545,Z 448.597,A -85,B 0,C 180,E1 -3564.333,E2 -3564.333} C_VEL
LIN {X 0,Y 544.775,Z 448.63,A -85,B 0,C 180,E1 -3566.988,E2 -3566.988} C_VEL
LIN {X 0,Y 544.757,Z 451.768,A -85,B 0,C 180,E1 -3569.812,E2 -3569.812} C_VEL
LIN {X 0,Y 544.777,Z 455.526,A -85,B 0,C 180,E1 -3573.158,E2 -3573.158} C_VEL
LIN {X 0,Y 544.652,Z 458.304,A -85,B 0,C 180,E1 -3575.612,E2 -3575.612} C_VEL
LIN {X 0,Y 544.652,Z 461.314,A -85,B 0,C 180,E1 -3578.29,E2 -3578.29} C_VEL
LIN {X 0,Y 544.613,Z 464.608,A -85,B 0,C 180,E1 -3581.179,E2 -3581.179} C_VEL
LIN {X 0,Y 544.623,Z 467.379,A -85,B 0,C 180,E1 -3583.507,E2 -3583.507} C_VEL
LIN {X 0,Y 544.606,Z 471.223,A -85,B 0,C 180,E1 -3586.568,E2 -3586.568} C_VEL
LIN {X 0,Y 544.606,Z 471.673,A -85,B 0,C 180,E1 -3586.924,E2 -3586.924} C_VEL
LIN {X 0,Y 546.123,Z 481.165,A -85,B 0,C 180,E1 -3587.198,E2 -3587.198} C_VEL
LIN {X 0,Y 545.923,Z 494.151,A -85,B 0,C 180,E1 -3587.642,E2 -3587.642} C_VEL
LIN {X 0,Y 545.712,Z 506.728,A -85,B 0,C 180,E1 -3588.237,E2 -3588.237} C_VEL
LIN {X 0,Y 545.556,Z 518.285,A -85,B 0,C 180,E1 -3588.952,E2 -3588.952} C_VEL
LIN {X 0,Y 545.287,Z 529.022,A -85,B 0,C 180,E1 -3589.792,E2 -3589.792} C_VEL
LIN {X 0,Y 545.123,Z 538.685,A -85,B 0,C 180,E1 -3590.726,E2 -3590.726} C_VEL
LIN {X 0,Y 544.975,Z 546.603,A -85,B 0,C 180,E1 -3591.658,E2 -3591.658} C_VEL
LIN {X 0,Y 544.83,Z 554.35,A -85,B 0,C 180,E1 -3592.775,E2 -3592.775} C_VEL
LIN {X 0,Y 544.778,Z 561.459,A -85,B 0,C 180,E1 -3594.076,E2 -3594.076} C_VEL
LIN {X 0,Y 544.629,Z 566.199,A -85,B 0,C 180,E1 -3595.188,E2 -3595.188} C_VEL
LIN {X 0,Y 544.669,Z 569.831,A -85,B 0,C 180,E1 -3596.301,E2 -3596.301} C_VEL
LIN {X 0,Y 544.651,Z 571.707,A -85,B 0,C 180,E1 -3597.041,E2 -3597.041} C_VEL
LIN {X 0,Y 544.571,Z 573.129,A -85,B 0,C 180,E1 -3597.781,E2 -3597.781} C_VEL
LIN {X 0,Y 544.543,Z 574.758,A -85,B 0,C 180,E1 -3599.26,E2 -3599.26} C_VEL
LIN {X 0,Y 544.541,Z 574.996,A -85,B 0,C 180,E1 -3600,E2 -3600} C_VEL
LIN {X 0,Y 544.542,Z 574.814,A -85,B 0,C 180,E1 -3600.739,E2 -3600.739} C_VEL
LIN {X 0,Y 544.57,Z 573.264,A -85,B 0,C 180,E1 -3602.219,E2 -3602.219} C_VEL
LIN {X 0,Y 544.651,Z 571.902,A -85,B 0,C 180,E1 -3602.959,E2 -3602.959} C_VEL
LIN {X 0,Y 544.684,Z 569.024,A -85,B 0,C 180,E1 -3604.069,E2 -3604.069} C_VEL
LIN {X 0,Y 544.653,Z 565.123,A -85,B 0,C 180,E1 -3605.182,E2 -3605.182} C_VEL
LIN {X 0,Y 544.726,Z 559.89,A -85,B 0,C 180,E1 -3606.337,E2 -3606.337} C_VEL
LIN {X 0,Y 544.859,Z 552.534,A -85,B 0,C 180,E1 -3607.597,E2 -3607.597} C_VEL
LIN {X 0,Y 544.999,Z 544.351,A -85,B 0,C 180,E1 -3608.715,E2 -3608.715} C_VEL
LIN {X 0,Y 545.159,Z 535.981,A -85,B 0,C 180,E1 -3609.648,E2 -3609.648} C_VEL
LIN {X 0,Y 545.379,Z 525.657,A -85,B 0,C 180,E1 -3610.581,E2 -3610.581} C_VEL
LIN {X 0,Y 545.634,Z 514.293,A -85,B 0,C 180,E1 -3611.403,E2 -3611.403} C_VEL
LIN {X 0,Y 545.772,Z 504.251,A -85,B 0,C 180,E1 -3611.984,E2 -3611.984} C_VEL
LIN {X 0,Y 545.968,Z 491.713,A -85,B 0,C 180,E1 -3612.546,E2 -3612.546} C_VEL
LIN {X 0,Y 545.957,Z 479.555,A -85,B 0,C 180,E1 -3612.938,E2 -3612.938} C_VEL
LIN {X 0,Y 544.594,Z 471.667,A -85,B 0,C 180,E1 -3613.171,E2 -3613.171} C_VEL
LIN {X 0,Y 544.592,Z 468.453,A -85,B 0,C 180,E1 -3615.724,E2 -3615.724} C_VEL
LIN {X 0,Y 544.605,Z 465.729,A -85,B 0,C 180,E1 -3618.042,E2 -3618.042} C_VEL
LIN {X 0,Y 544.673,Z 463.305,A -85,B 0,C 180,E1 -3620.389,E2 -3620.389} C_VEL
LIN {X 0,Y 544.741,Z 460.007,A -85,B 0,C 180,E1 -3623.575,E2 -3623.575} C_VEL
LIN {X 0,Y 544.775,Z 457.545,A -85,B 0,C 180,E1 -3626.016,E2 -3626.016} C_VEL
LIN {X 0,Y 544.873,Z 454.892,A -85,B 0,C 180,E1 -3628.706,E2 -3628.706} C_VEL
LIN {X 0,Y 544.951,Z 451.936,A -85,B 0,C 180,E1 -3631.66,E2 -3631.66} C_VEL
LIN {X 0,Y 545.005,Z 449.207,A -85,B 0,C 180,E1 -3634.569,E2 -3634.569} C_VEL
LIN {X 0,Y 544.999,Z 448.601,A -85,B 0,C 180,E1 -3635.667,E2 -3635.667} C_VEL
LIN {X 0,Y 545.056,Z 448.593,A -85,B 0,C 180,E1 -3638.237,E2 -3638.237} C_VEL
LIN {X 0,Y 545.091,Z 448.589,A -85,B 0,C 180,E1 -3641.114,E2 -3641.114} C_VEL
LIN {X 0,Y 545.062,Z 448.593,A -85,B 0,C 180,E1 -3644.129,E2 -3644.129} C_VEL
LIN {X 0,Y 545.081,Z 448.59,A -85,B 0,C 180,E1 -3646.893,E2 -3646.893} C_VEL
LIN {X 0,Y 545.078,Z 448.592,A -85,B 0,C 180,E1 -3649.858,E2 -3649.858} C_VEL
LIN {X 0,Y 545.128,Z 448.74,A -85,B 0,C 180,E1 -3651.415,E2 -3651.415} C_VEL
LIN {X 0,Y 545.9,Z 453.136,A -85,B 0,C 180,E1 -3653.686,E2 -3653.686} C_VEL
LIN {X 0,Y 545.999,Z 456.349,A -85,B 0,C 180,E1 -3655.055,E2 -3655.055} C_VEL
LIN {X 0,Y 545.696,Z 463.423,A -85,B 0,C 180,E1 -3657.691,E2 -3657.691} C_VEL
LIN {X 0,Y 545.462,Z 471.022,A -85,B 0,C 180,E1 -3660.261,E2 -3660.261} C_VEL
LIN {X 0,Y 545.333,Z 480.45,A -85,B 0,C 180,E1 -3663.188,E2 -3663.188} C_VEL
LIN {X 0,Y 545.21,Z 489.883,A -85,B 0,C 180,E1 -3665.977,E2 -3665.977} C_VEL
LIN {X 0,Y 545.126,Z 499.835,A -85,B 0,C 180,E1 -3668.839,E2 -3668.839} C_VEL
LIN {X 0,Y 545.03,Z 509.492,A -85,B 0,C 180,E1 -3671.583,E2 -3671.583} C_VEL
LIN {X 0,Y 544.928,Z 520.083,A -85,B 0,C 180,E1 -3674.669,E2 -3674.669} C_VEL
LIN {X 0,Y 544.825,Z 527.53,A -85,B 0,C 180,E1 -3676.811,E2 -3676.811} C_VEL
LIN {X 0,Y 546.149,Z 536.515,A -85,B 0,C 180,E1 -3677.033,E2 -3677.033} C_VEL
LIN {X 0,Y 546.01,Z 549.171,A -85,B 0,C 180,E1 -3677.408,E2 -3677.408} C_VEL
LIN {X 0,Y 545.847,Z 561.489,A -85,B 0,C 180,E1 -3677.923,E2 -3677.923} C_VEL
LIN {X 0,Y 545.62,Z 573.337,A -85,B 0,C 180,E1 -3678.579,E2 -3678.579} C_VEL
LIN {X 0,Y 545.409,Z 585.093,A -85,B 0,C 180,E1 -3679.419,E2 -3679.419} C_VEL
LIN {X 0,Y 545.165,Z 595.538,A -85,B 0,C 180,E1 -3680.352,E2 -3680.352} C_VEL
LIN {X 0,Y 545.029,Z 603.99,A -85,B 0,C 180,E1 -3681.285,E2 -3681.285} C_VEL
LIN {X 0,Y 544.859,Z 612.235,A -85,B 0,C 180,E1 -3682.402,E2 -3682.402} C_VEL
LIN {X 0,Y 544.734,Z 619.615,A -85,B 0,C 180,E1 -3683.655,E2 -3683.655} C_VEL
LIN {X 0,Y 544.654,Z 624.949,A -85,B 0,C 180,E1 -3684.818,E2 -3684.818} C_VEL
LIN {X 0,Y 544.683,Z 628.894,A -85,B 0,C 180,E1 -3685.93,E2 -3685.93} C_VEL
LIN {X 0,Y 544.65,Z 631.807,A -85,B 0,C 180,E1 -3687.041,E2 -3687.041} C_VEL
LIN {X 0,Y 544.546,Z 634.184,A -85,B 0,C 180,E1 -3688.521,E2 -3688.521} C_VEL
LIN {X 0,Y 544.541,Z 635,A -85,B 0,C 180,E1 -3690,E2 -3690} C_VEL
LIN {X 0,Y 544.546,Z 634.185,A -85,B 0,C 180,E1 -3691.479,E2 -3691.479} C_VEL
LIN {X 0,Y 544.65,Z 631.81,A -85,B 0,C 180,E1 -3692.959,E2 -3692.959} C_VEL
LIN {X 0,Y 544.683,Z 628.896,A -85,B 0,C 180,E1 -3694.069,E2 -3694.069} C_VEL
LIN {X 0,Y 544.654,Z 624.949,A -85,B 0,C 180,E1 -3695.182,E2 -3695.182} C_VEL
LIN {X 0,Y 544.739,Z 619.704,A -85,B 0,C 180,E1 -3696.328,E2 -3696.328} C_VEL
LIN {X 0,Y 544.836,Z 613.468,A -85,B 0,C 180,E1 -3697.411,E2 -3697.411} C_VEL
LIN {X 0,Y 545.006,Z 605.478,A -85,B 0,C 180,E1 -3698.528,E2 -3698.528} C_VEL
LIN {X 0,Y 545.142,Z 597.335,A -85,B 0,C 180,E1 -3699.461,E2 -3699.461} C_VEL
LIN {X 0,Y 545.364,Z 587.399,A -85,B 0,C 180,E1 -3700.394,E2 -3700.394} C_VEL
LIN {X 0,Y 545.561,Z 576.593,A -85,B 0,C 180,E1 -3701.208,E2 -3701.208} C_VEL
LIN {X 0,Y 545.741,Z 565.174,A -85,B 0,C 180,E1 -3701.891,E2 -3701.891} C_VEL
LIN {X 0,Y 545.943,Z 552.976,A -85,B 0,C 180,E1 -3702.452,E2 -3702.452} C_VEL
LIN {X 0,Y 546.125,Z 540.176,A -85,B 0,C 180,E1 -3702.873,E2 -3702.873} C_VEL
LIN {X 0,Y 545.913,Z 534.364,A -85,B 0,C 180,E1 -3703.02,E2 -3703.02} C_VEL
LIN {X 0,Y 544.825,Z 527.53,A -85,B 0,C 180,E1 -3703.189,E2 -3703.189} C_VEL
LIN {X 0,Y 544.938,Z 517.436,A -85,B 0,C 180,E1 -3706.098,E2 -3706.098} C_VEL
LIN {X 0,Y 545.068,Z 506.837,A -85,B 0,C 180,E1 -3709.195,E2 -3709.195} C_VEL
LIN {X 0,Y 545.173,Z 497.258,A -85,B 0,C 180,E1 -3711.953,E2 -3711.953} C_VEL
LIN {X 0,Y 545.305,Z 487.944,A -85,B 0,C 180,E1 -3714.763,E2 -3714.763} C_VEL
LIN {X 0,Y 545.517,Z 478.617,A -85,B 0,C 180,E1 -3717.632,E2 -3717.632} C_VEL
LIN {X 0,Y 545.708,Z 468.011,A -85,B 0,C 180,E1 -3721.007,E2 -3721.007} C_VEL
LIN {X 0,Y 545.956,Z 458.876,A -85,B 0,C 180,E1 -3724.054,E2 -3724.054} C_VEL
LIN {X 0,Y 545.94,Z 453.842,A -85,B 0,C 180,E1 -3725.805,E2 -3725.805} C_VEL
LIN {X 0,Y 545.056,Z 448.594,A -85,B 0,C 180,E1 -3727.768,E2 -3727.768} C_VEL
LIN {X 0,Y 545.094,Z 448.586,A -85,B 0,C 180,E1 -3730.474,E2 -3730.474} C_VEL
LIN {X 0,Y 545.08,Z 448.591,A -85,B 0,C 180,E1 -3733.107,E2 -3733.107} C_VEL
LIN {X 0,Y 545.067,Z 448.592,A -85,B 0,C 180,E1 -3736.224,E2 -3736.224} C_VEL
LIN {X 0,Y 545.09,Z 448.587,A -85,B 0,C 180,E1 -3738.886,E2 -3738.886} C_VEL
LIN {X 0,Y 545.053,Z 448.589,A -85,B 0,C 180,E1 -3741.763,E2 -3741.763} C_VEL
LIN {X 0,Y 545.039,Z 448.592,A -85,B 0,C 180,E1 -3744.532,E2 -3744.532} C_VEL
LIN {X 0,Y 545.071,Z 448.59,A -85,B 0,C 180,E1 -3747.212,E2 -3747.212} C_VEL
LIN {X 0,Y 545.066,Z 448.59,A -85,B 0,C 180,E1 -3749.811,E2 -3749.811} C_VEL
LIN {X 0,Y 545.092,Z 448.585,A -85,B 0,C 180,E1 -3752.344,E2 -3752.344} C_VEL
LIN {X 0,Y 545.12,Z 448.586,A -85,B 0,C 180,E1 -3754.821,E2 -3754.821} C_VEL
LIN {X 0,Y 545.041,Z 448.591,A -85,B 0,C 180,E1 -3757.242,E2 -3757.242} C_VEL
LIN {X 0,Y 545.123,Z 448.581,A -85,B 0,C 180,E1 -3760.415,E2 -3760.415} C_VEL
LIN {X 0,Y 545.076,Z 448.586,A -85,B 0,C 180,E1 -3763.521,E2 -3763.521} C_VEL
LIN {X 0,Y 545.098,Z 448.589,A -85,B 0,C 180,E1 -3765.82,E2 -3765.82} C_VEL
LIN {X 0,Y 545.121,Z 448.586,A -85,B 0,C 180,E1 -3768.849,E2 -3768.849} C_VEL
LIN {X 0,Y 545.131,Z 448.583,A -85,B 0,C 180,E1 -3771.847,E2 -3771.847} C_VEL
LIN {X 0,Y 545.207,Z 448.573,A -85,B 0,C 180,E1 -3774.823,E2 -3774.823} C_VEL
LIN {X 0,Y 545.196,Z 448.572,A -85,B 0,C 180,E1 -3777.784,E2 -3777.784} C_VEL
LIN {X 0,Y 545.217,Z 448.57,A -85,B 0,C 180,E1 -3780.739,E2 -3780.739} C_VEL
LIN {X 0,Y 545.176,Z 448.578,A -85,B 0,C 180,E1 -3782.956,E2 -3782.956} C_VEL
LIN {X 0,Y 545.172,Z 448.578,A -85,B 0,C 180,E1 -3785.92,E2 -3785.92} C_VEL
LIN {X 0,Y 545.123,Z 448.584,A -85,B 0,C 180,E1 -3788.9,E2 -3788.9} C_VEL
LIN {X 0,Y 545.138,Z 448.58,A -85,B 0,C 180,E1 -3791.904,E2 -3791.904} C_VEL
LIN {X 0,Y 545.089,Z 448.587,A -85,B 0,C 180,E1 -3794.944,E2 -3794.944} C_VEL
LIN {X 0,Y 545.081,Z 448.587,A -85,B 0,C 180,E1 -3798.026,E2 -3798.026} C_VEL
LIN {X 0,Y 545.099,Z 448.586,A -85,B 0,C 180,E1 -3800.372,E2 -3800.372} C_VEL
LIN {X 0,Y 545.084,Z 448.587,A -85,B 0,C 180,E1 -3803.559,E2 -3803.559} C_VEL
LIN {X 0,Y 545.083,Z 448.588,A -85,B 0,C 180,E1 -3806.001,E2 -3806.001} C_VEL
LIN {X 0,Y 545.093,Z 448.585,A -85,B 0,C 180,E1 -3808.748,E2 -3808.748} C_VEL
LIN {X 0,Y 545.062,Z 448.588,A -85,B 0,C 180,E1 -3811.679,E2 -3811.679} C_VEL
LIN {X 0,Y 545.08,Z 448.587,A -85,B 0,C 180,E1 -3814.564,E2 -3814.564} C_VEL
LIN {X 0,Y 545.069,Z 448.59,A -85,B 0,C 180,E1 -3817.008,E2 -3817.008} C_VEL
LIN {X 0,Y 544.36,Z 448.68,A -85,B 0,C 180,E1 -3817.624,E2 -3817.624} C_VEL
LIN {X 0,Y 541.493,Z 449.037,A -85,B 0,C 180,E1 -3818.625,E2 -3818.625} C_VEL
LIN {X 0,Y 539.105,Z 449.331,A -85,B 0,C 180,E1 -3819.431,E2 -3819.431} C_VEL
LIN {X 0,Y 538.095,Z 449.458,A -85,B 0,C 180,E1 -3820.053,E2 -3820.053} C_VEL
LIN {X 0,Y 538.02,Z 449.464,A -85,B 0,C 180,E1 -3820.263,E2 -3820.263} C_VEL
LIN {X 0,Y 538.037,Z 449.465,A -85,B 0,C 180,E1 -3822.989,E2 -3822.989} C_VEL
LIN {X 0,Y 538.034,Z 449.464,A -85,B 0,C 180,E1 -3825.926,E2 -3825.926} C_VEL
LIN {X 0,Y 538.052,Z 449.463,A -85,B 0,C 180,E1 -3829.253,E2 -3829.253} C_VEL
LIN {X 0,Y 537.996,Z 449.469,A -85,B 0,C 180,E1 -3832.123,E2 -3832.123} C_VEL
LIN {X 0,Y 538.017,Z 449.466,A -85,B 0,C 180,E1 -3834.917,E2 -3834.917} C_VEL
LIN {X 0,Y 538.023,Z 449.47,A -85,B 0,C 180,E1 -3837.618,E2 -3837.618} C_VEL
LIN {X 0,Y 538.021,Z 449.467,A -85,B 0,C 180,E1 -3840.239,E2 -3840.239} C_VEL
LIN {X 0,Y 538.055,Z 449.461,A -85,B 0,C 180,E1 -3842.796,E2 -3842.796} C_VEL
LIN {X 0,Y 538.053,Z 449.466,A -85,B 0,C 180,E1 -3845.293,E2 -3845.293} C_VEL
LIN {X 0,Y 538.027,Z 449.468,A -85,B 0,C 180,E1 -3848.546,E2 -3848.546} C_VEL
LIN {X 0,Y 538.038,Z 449.464,A -85,B 0,C 180,E1 -3850.94,E2 -3850.94} C_VEL
LIN {X 0,Y 538.023,Z 449.469,A -85,B 0,C 180,E1 -3853.299,E2 -3853.299} C_VEL
LIN {X 0,Y 538.069,Z 449.46,A -85,B 0,C 180,E1 -3855.631,E2 -3855.631} C_VEL
LIN {X 0,Y 538.083,Z 449.458,A -85,B 0,C 180,E1 -3858.702,E2 -3858.702} C_VEL
LIN {X 0,Y 538.09,Z 449.457,A -85,B 0,C 180,E1 -3861.74,E2 -3861.74} C_VEL
LIN {X 0,Y 538.162,Z 449.447,A -85,B 0,C 180,E1 -3864.755,E2 -3864.755} C_VEL
LIN {X 0,Y 538.173,Z 449.447,A -85,B 0,C 180,E1 -3867.755,E2 -3867.755} C_VEL
LIN {X 0,Y 538.186,Z 449.445,A -85,B 0,C 180,E1 -3870.748,E2 -3870.748} C_VEL
LIN {X 0,Y 538.141,Z 449.452,A -85,B 0,C 180,E1 -3872.995,E2 -3872.995} C_VEL
LIN {X 0,Y 538.13,Z 449.453,A -85,B 0,C 180,E1 -3875.997,E2 -3875.997} C_VEL
LIN {X 0,Y 538.067,Z 449.459,A -85,B 0,C 180,E1 -3879.018,E2 -3879.018} C_VEL
LIN {X 0,Y 538.089,Z 449.458,A -85,B 0,C 180,E1 -3882.063,E2 -3882.063} C_VEL
LIN {X 0,Y 538.05,Z 449.461,A -85,B 0,C 180,E1 -3885.144,E2 -3885.144} C_VEL
LIN {X 0,Y 538.034,Z 449.464,A -85,B 0,C 180,E1 -3888.27,E2 -3888.27} C_VEL
LIN {X 0,Y 538.043,Z 449.466,A -85,B 0,C 180,E1 -3890.651,E2 -3890.651} C_VEL
LIN {X 0,Y 538.01,Z 449.47,A -85,B 0,C 180,E1 -3893.888,E2 -3893.888} C_VEL
LIN {X 0,Y 538.047,Z 449.464,A -85,B 0,C 180,E1 -3896.367,E2 -3896.367} C_VEL
LIN {X 0,Y 538.036,Z 449.464,A -85,B 0,C 180,E1 -3898.933,E2 -3898.933} C_VEL
LIN {X 0,Y 538.015,Z 449.468,A -85,B 0,C 180,E1 -3901.887,E2 -3901.887} C_VEL
LIN {X 0,Y 538.018,Z 449.47,A -85,B 0,C 180,E1 -3904.618,E2 -3904.618} C_VEL
LIN {X 0,Y 538.009,Z 449.467,A -85,B 0,C 180,E1 -3907.17,E2 -3907.17} C_VEL
LIN {X 0,Y 538.03,Z 449.465,A -85,B 0,C 180,E1 -3909.797,E2 -3909.797} C_VEL
LIN {X 0,Y 538.024,Z 449.466,A -85,B 0,C 180,E1 -3912.786,E2 -3912.786} C_VEL
LIN {X 0,Y 538.034,Z 449.465,A -85,B 0,C 180,E1 -3915.925,E2 -3915.925} C_VEL
LIN {X 0,Y 538.054,Z 449.462,A -85,B 0,C 180,E1 -3919.253,E2 -3919.253} C_VEL
LIN {X 0,Y 537.995,Z 449.47,A -85,B 0,C 180,E1 -3922.122,E2 -3922.122} C_VEL
LIN {X 0,Y 537.939,Z 449.48,A -85,B 0,C 180,E1 -3924.911,E2 -3924.911} C_VEL
LIN {X 0,Y 537.762,Z 449.503,A -85,B 0,C 180,E1 -3926.764,E2 -3926.764} C_VEL
LIN {X 0,Y 537.696,Z 450.558,A -85,B 0,C 180,E1 -3928.167,E2 -3928.167} C_VEL
LIN {X 0,Y 537.65,Z 453.861,A -85,B 0,C 180,E1 -3931.141,E2 -3931.141} C_VEL
LIN {X 0,Y 537.671,Z 456.622,A -85,B 0,C 180,E1 -3933.613,E2 -3933.613} C_VEL
LIN {X 0,Y 537.621,Z 459.558,A -85,B 0,C 180,E1 -3936.216,E2 -3936.216} C_VEL
LIN {X 0,Y 537.578,Z 462.161,A -85,B 0,C 180,E1 -3938.527,E2 -3938.527} C_VEL
LIN {X 0,Y 537.533,Z 464.83,A -85,B 0,C 180,E1 -3940.921,E2 -3940.921} C_VEL
LIN {X 0,Y 537.548,Z 467.507,A -85,B 0,C 180,E1 -3943.284,E2 -3943.284} C_VEL
LIN {X 0,Y 537.515,Z 471.223,A -85,B 0,C 180,E1 -3946.388,E2 -3946.388} C_VEL
LIN {X 0,Y 537.488,Z 471.674,A -85,B 0,C 180,E1 -3946.748,E2 -3946.748} C_VEL
LIN {X 0,Y 539.213,Z 482.008,A -85,B 0,C 180,E1 -3947.055,E2 -3947.055} C_VEL
LIN {X 0,Y 539.003,Z 494.164,A -85,B 0,C 180,E1 -3947.48,E2 -3947.48} C_VEL
LIN {X 0,Y 538.76,Z 506.307,A -85,B 0,C 180,E1 -3948.059,E2 -3948.059} C_VEL
LIN {X 0,Y 538.58,Z 518.292,A -85,B 0,C 180,E1 -3948.807,E2 -3948.807} C_VEL
LIN {X 0,Y 538.274,Z 529.027,A -85,B 0,C 180,E1 -3949.658,E2 -3949.658} C_VEL
LIN {X 0,Y 538.086,Z 538.69,A -85,B 0,C 180,E1 -3950.603,E2 -3950.603} C_VEL
LIN {X 0,Y 537.923,Z 546.608,A -85,B 0,C 180,E1 -3951.548,E2 -3951.548} C_VEL
LIN {X 0,Y 537.76,Z 554.354,A -85,B 0,C 180,E1 -3952.679,E2 -3952.679} C_VEL
LIN {X 0,Y 537.694,Z 561.462,A -85,B 0,C 180,E1 -3953.998,E2 -3953.998} C_VEL
LIN {X 0,Y 537.54,Z 566.201,A -85,B 0,C 180,E1 -3955.125,E2 -3955.125} C_VEL
LIN {X 0,Y 537.591,Z 569.832,A -85,B 0,C 180,E1 -3956.252,E2 -3956.252} C_VEL
LIN {X 0,Y 537.551,Z 571.709,A -85,B 0,C 180,E1 -3957.002,E2 -3957.002} C_VEL
LIN {X 0,Y 537.489,Z 573.129,A -85,B 0,C 180,E1 -3957.752,E2 -3957.752} C_VEL
LIN {X 0,Y 537.443,Z 574.758,A -85,B 0,C 180,E1 -3959.251,E2 -3959.251} C_VEL
LIN {X 0,Y 537.442,Z 574.996,A -85,B 0,C 180,E1 -3960,E2 -3960} C_VEL
LIN {X 0,Y 537.442,Z 574.814,A -85,B 0,C 180,E1 -3960.749,E2 -3960.749} C_VEL
LIN {X 0,Y 537.489,Z 573.262,A -85,B 0,C 180,E1 -3962.248,E2 -3962.248} C_VEL
LIN {X 0,Y 537.552,Z 571.901,A -85,B 0,C 180,E1 -3962.998,E2 -3962.998} C_VEL
LIN {X 0,Y 537.603,Z 569.023,A -85,B 0,C 180,E1 -3964.123,E2 -3964.123} C_VEL
LIN {X 0,Y 537.587,Z 565.12,A -85,B 0,C 180,E1 -3965.251,E2 -3965.251} C_VEL
LIN {X 0,Y 537.64,Z 560.36,A -85,B 0,C 180,E1 -3966.322,E2 -3966.322} C_VEL
LIN {X 0,Y 537.79,Z 553.757,A -85,B 0,C 180,E1 -3967.509,E2 -3967.509} C_VEL
LIN {X 0,Y 537.952,Z 545.831,A -85,B 0,C 180,E1 -3968.641,E2 -3968.641} C_VEL
LIN {X 0,Y 538.132,Z 535.975,A -85,B 0,C 180,E1 -3969.775,E2 -3969.775} C_VEL
LIN {X 0,Y 538.375,Z 525.648,A -85,B 0,C 180,E1 -3970.721,E2 -3970.721} C_VEL
LIN {X 0,Y 538.651,Z 514.706,A -85,B 0,C 180,E1 -3971.525,E2 -3971.525} C_VEL
LIN {X 0,Y 538.824,Z 504.239,A -85,B 0,C 180,E1 -3972.141,E2 -3972.141} C_VEL
LIN {X 0,Y 539.01,Z 492.915,A -85,B 0,C 180,E1 -3972.663,E2 -3972.663} C_VEL
LIN {X 0,Y 539.064,Z 480.53,A -85,B 0,C 180,E1 -3973.081,E2 -3973.081} C_VEL
LIN {X 0,Y 537.524,Z 471.666,A -85,B 0,C 180,E1 -3973.347,E2 -3973.347} C_VEL
LIN {X 0,Y 537.516,Z 468.674,A -85,B 0,C 180,E1 -3975.937,E2 -3975.937} C_VEL
LIN {X 0,Y 537.541,Z 466.2,A -85,B 0,C 180,E1 -3978.287,E2 -3978.287} C_VEL
LIN {X 0,Y 537.62,Z 463.782,A -85,B 0,C 180,E1 -3980.668,E2 -3980.668} C_VEL
LIN {X 0,Y 537.686,Z 460.443,A -85,B 0,C 180,E1 -3983.903,E2 -3983.903} C_VEL
LIN {X 0,Y 537.742,Z 457.964,A -85,B 0,C 180,E1 -3986.383,E2 -3986.383} C_VEL
LIN {X 0,Y 537.815,Z 455.506,A -85,B 0,C 180,E1 -3988.915,E2 -3988.915} C_VEL
LIN {X 0,Y 537.897,Z 452.64,A -85,B 0,C 180,E1 -3991.867,E2 -3991.867} C_VEL
LIN {X 0,Y 537.969,Z 450.15,A -85,B 0,C 180,E1 -3994.61,E2 -3994.61} C_VEL
LIN {X 0,Y 537.961,Z 449.478,A -85,B 0,C 180,E1 -3996.007,E2 -3996.007} C_VEL
LIN {X 0,Y 538.017,Z 449.471,A -85,B 0,C 180,E1 -3998.83,E2 -3998.83} C_VEL
LIN {X 0,Y 538.038,Z 449.467,A -85,B 0,C 180,E1 -4001.879,E2 -4001.879} C_VEL
LIN {X 0,Y 538.036,Z 449.469,A -85,B 0,C 180,E1 -4005.141,E2 -4005.141} C_VEL
LIN {X 0,Y 538.038,Z 449.468,A -85,B 0,C 180,E1 -4008.227,E2 -4008.227} C_VEL
LIN {X 0,Y 538.061,Z 449.569,A -85,B 0,C 180,E1 -4010.933,E2 -4010.933} C_VEL
LIN {X 0,Y 538.746,Z 453.499,A -85,B 0,C 180,E1 -4013.124,E2 -4013.124} C_VEL
LIN {X 0,Y 539.063,Z 456.558,A -85,B 0,C 180,E1 -4014.538,E2 -4014.538} C_VEL
LIN {X 0,Y 538.76,Z 462.186,A -85,B 0,C 180,E1 -4016.778,E2 -4016.778} C_VEL
LIN {X 0,Y 538.524,Z 469.78,A -85,B 0,C 180,E1 -4019.467,E2 -4019.467} C_VEL
LIN {X 0,Y 538.337,Z 480.098,A -85,B 0,C 180,E1 -4022.811,E2 -4022.811} C_VEL
LIN {X 0,Y 538.172,Z 489.715,A -85,B 0,C 180,E1 -4025.71,E2 -4025.71} C_VEL
LIN {X 0,Y 538.069,Z 499.363,A -85,B 0,C 180,E1 -4028.548,E2 -4028.548} C_VEL
LIN {X 0,Y 537.966,Z 509.183,A -85,B 0,C 180,E1 -4031.333,E2 -4031.333} C_VEL
LIN {X 0,Y 537.876,Z 518.759,A -85,B 0,C 180,E1 -4034.074,E2 -4034.074} C_VEL
LIN {X 0,Y 537.754,Z 527.53,A -85,B 0,C 180,E1 -4036.634,E2 -4036.634} C_VEL
LIN {X 0,Y 539.223,Z 537.43,A -85,B 0,C 180,E1 -4036.887,E2 -4036.887} C_VEL
LIN {X 0,Y 539.083,Z 550.471,A -85,B 0,C 180,E1 -4037.291,E2 -4037.291} C_VEL
LIN {X 0,Y 538.891,Z 561.487,A -85,B 0,C 180,E1 -4037.765,E2 -4037.765} C_VEL
LIN {X 0,Y 538.652,Z 573.657,A -85,B 0,C 180,E1 -4038.45,E2 -4038.45} C_VEL
LIN {X 0,Y 538.382,Z 585.092,A -85,B 0,C 180,E1 -4039.279,E2 -4039.279} C_VEL
LIN {X 0,Y 538.138,Z 595.538,A -85,B 0,C 180,E1 -4040.225,E2 -4040.225} C_VEL
LIN {X 0,Y 537.974,Z 603.991,A -85,B 0,C 180,E1 -4041.17,E2 -4041.17} C_VEL
LIN {X 0,Y 537.817,Z 612.235,A -85,B 0,C 180,E1 -4042.302,E2 -4042.302} C_VEL
LIN {X 0,Y 537.683,Z 618.749,A -85,B 0,C 180,E1 -4043.409,E2 -4043.409} C_VEL
LIN {X 0,Y 537.676,Z 623.365,A -85,B 0,C 180,E1 -4044.374,E2 -4044.374} C_VEL
LIN {X 0,Y 537.558,Z 627.677,A -85,B 0,C 180,E1 -4045.501,E2 -4045.501} C_VEL
LIN {X 0,Y 537.591,Z 629.958,A -85,B 0,C 180,E1 -4046.252,E2 -4046.252} C_VEL
LIN {X 0,Y 537.551,Z 631.807,A -85,B 0,C 180,E1 -4047.002,E2 -4047.002} C_VEL
LIN {X 0,Y 537.451,Z 634.183,A -85,B 0,C 180,E1 -4048.501,E2 -4048.501} C_VEL
LIN {X 0,Y 537.442,Z 635,A -85,B 0,C 180,E1 -4050,E2 -4050} C_VEL
LIN {X 0,Y 537.451,Z 634.185,A -85,B 0,C 180,E1 -4051.499,E2 -4051.499} C_VEL
LIN {X 0,Y 537.551,Z 631.81,A -85,B 0,C 180,E1 -4052.998,E2 -4052.998} C_VEL
LIN {X 0,Y 537.603,Z 628.896,A -85,B 0,C 180,E1 -4054.123,E2 -4054.123} C_VEL
LIN {X 0,Y 537.588,Z 624.949,A -85,B 0,C 180,E1 -4055.251,E2 -4055.251} C_VEL
LIN {X 0,Y 537.65,Z 620.08,A -85,B 0,C 180,E1 -4056.335,E2 -4056.335} C_VEL
LIN {X 0,Y 537.79,Z 613.467,A -85,B 0,C 180,E1 -4057.509,E2 -4057.509} C_VEL
LIN {X 0,Y 537.972,Z 605.478,A -85,B 0,C 180,E1 -4058.64,E2 -4058.64} C_VEL
LIN {X 0,Y 538.118,Z 597.334,A -85,B 0,C 180,E1 -4059.585,E2 -4059.585} C_VEL
LIN {X 0,Y 538.361,Z 587.398,A -85,B 0,C 180,E1 -4060.531,E2 -4060.531} C_VEL
LIN {X 0,Y 538.573,Z 577.591,A -85,B 0,C 180,E1 -4061.288,E2 -4061.288} C_VEL
LIN {X 0,Y 538.763,Z 566.442,A -85,B 0,C 180,E1 -4061.978,E2 -4061.978} C_VEL
LIN {X 0,Y 538.995,Z 554.104,A -85,B 0,C 180,E1 -4062.567,E2 -4062.567} C_VEL
LIN {X 0,Y 539.195,Z 541.088,A -85,B 0,C 180,E1 -4063.017,E2 -4063.017} C_VEL
LIN {X 0,Y 538.975,Z 534.933,A -85,B 0,C 180,E1 -4063.179,E2 -4063.179} C_VEL
LIN {X 0,Y 537.754,Z 527.53,A -85,B 0,C 180,E1 -4063.365,E2 -4063.365} C_VEL
LIN {X 0,Y 537.875,Z 518.759,A -85,B 0,C 180,E1 -4065.926,E2 -4065.926} C_VEL
LIN {X 0,Y 537.966,Z 509.311,A -85,B 0,C 180,E1 -4068.667,E2 -4068.667} C_VEL
LIN {X 0,Y 538.092,Z 499.741,A -85,B 0,C 180,E1 -4071.451,E2 -4071.451} C_VEL
LIN {X 0,Y 538.241,Z 490.448,A -85,B 0,C 180,E1 -4074.286,E2 -4074.286} C_VEL
LIN {X 0,Y 538.452,Z 480.333,A -85,B 0,C 180,E1 -4077.432,E2 -4077.432} C_VEL
LIN {X 0,Y 538.697,Z 470.552,A -85,B 0,C 180,E1 -4080.584,E2 -4080.584} C_VEL
LIN {X 0,Y 538.92,Z 462.091,A -85,B 0,C 180,E1 -4083.424,E2 -4083.424} C_VEL
LIN {X 0,Y 539.018,Z 456.252,A -85,B 0,C 180,E1 -4085.466,E2 -4085.466} C_VEL
LIN {X 0,Y 538.416,Z 451.505,A -85,B 0,C 180,E1 -4087.227,E2 -4087.227} C_VEL
LIN {X 0,Y 538.026,Z 449.47,A -85,B 0,C 180,E1 -4088.068,E2 -4088.068} C_VEL
LIN {X 0,Y 538.053,Z 449.463,A -85,B 0,C 180,E1 -4090.775,E2 -4090.775} C_VEL
LIN {X 0,Y 538.032,Z 449.465,A -85,B 0,C 180,E1 -4094.075,E2 -4094.075} C_VEL
LIN {X 0,Y 538.026,Z 449.466,A -85,B 0,C 180,E1 -4097.215,E2 -4097.215} C_VEL
LIN {X 0,Y 538.024,Z 449.465,A -85,B 0,C 180,E1 -4100.203,E2 -4100.203} C_VEL
LIN {X 0,Y 538.026,Z 449.465,A -85,B 0,C 180,E1 -4103.067,E2 -4103.067} C_VEL
LIN {X 0,Y 538.021,Z 449.467,A -85,B 0,C 180,E1 -4105.827,E2 -4105.827} C_VEL
LIN {X 0,Y 538.011,Z 449.471,A -85,B 0,C 180,E1 -4108.499,E2 -4108.499} C_VEL
LIN {X 0,Y 538.062,Z 449.461,A -85,B 0,C 180,E1 -4111.1,E2 -4111.1} C_VEL
LIN {X 0,Y 538.044,Z 449.464,A -85,B 0,C 180,E1 -4113.633,E2 -4113.633} C_VEL
LIN {X 0,Y 538.009,Z 449.469,A -85,B 0,C 180,E1 -4116.122,E2 -4116.122} C_VEL
LIN {X 0,Y 538.042,Z 449.467,A -85,B 0,C 180,E1 -4119.349,E2 -4119.349} C_VEL
LIN {X 0,Y 538.057,Z 449.465,A -85,B 0,C 180,E1 -4122.517,E2 -4122.517} C_VEL
LIN {X 0,Y 538.067,Z 449.464,A -85,B 0,C 180,E1 -4125.631,E2 -4125.631} C_VEL
LIN {X 0,Y 538.08,Z 449.462,A -85,B 0,C 180,E1 -4128.702,E2 -4128.702} C_VEL
LIN {X 0,Y 538.088,Z 449.46,A -85,B 0,C 180,E1 -4131.74,E2 -4131.74} C_VEL
LIN {X 0,Y 538.165,Z 449.45,A -85,B 0,C 180,E1 -4134.755,E2 -4134.755} C_VEL
LIN {X 0,Y 538.168,Z 449.447,A -85,B 0,C 180,E1 -4137.755,E2 -4137.755} C_VEL
LIN {X 0,Y 538.187,Z 449.446,A -85,B 0,C 180,E1 -4140.748,E2 -4140.748} C_VEL
LIN {X 0,Y 538.142,Z 449.454,A -85,B 0,C 180,E1 -4142.995,E2 -4142.995} C_VEL
LIN {X 0,Y 538.126,Z 449.457,A -85,B 0,C 180,E1 -4145.997,E2 -4145.997} C_VEL
LIN {X 0,Y 538.074,Z 449.464,A -85,B 0,C 180,E1 -4149.018,E2 -4149.018} C_VEL
LIN {X 0,Y 538.086,Z 449.46,A -85,B 0,C 180,E1 -4152.063,E2 -4152.063} C_VEL
LIN {X 0,Y 538.049,Z 449.466,A -85,B 0,C 180,E1 -4155.144,E2 -4155.144} C_VEL
LIN {X 0,Y 538.033,Z 449.467,A -85,B 0,C 180,E1 -4158.27,E2 -4158.27} C_VEL
LIN {X 0,Y 538.043,Z 449.463,A -85,B 0,C 180,E1 -4160.651,E2 -4160.651} C_VEL
LIN {X 0,Y 538.007,Z 449.467,A -85,B 0,C 180,E1 -4163.888,E2 -4163.888} C_VEL
LIN {X 0,Y 538.045,Z 449.467,A -85,B 0,C 180,E1 -4166.367,E2 -4166.367} C_VEL
LIN {X 0,Y 538.034,Z 449.465,A -85,B 0,C 180,E1 -4168.934,E2 -4168.934} C_VEL
LIN {X 0,Y 538.018,Z 449.466,A -85,B 0,C 180,E1 -4171.888,E2 -4171.888} C_VEL
LIN {X 0,Y 538.03,Z 449.465,A -85,B 0,C 180,E1 -4174.62,E2 -4174.62} C_VEL
LIN {X 0,Y 538.011,Z 449.471,A -85,B 0,C 180,E1 -4177.171,E2 -4177.171} C_VEL
LIN {X 0,Y 538.02,Z 449.464,A -85,B 0,C 180,E1 -4180.263,E2 -4180.263} C_VEL
LIN {X 0,Y 537.373,Z 449.547,A -85,B 0,C 180,E1 -4180.889,E2 -4180.889} C_VEL
LIN {X 0,Y 534.526,Z 449.907,A -85,B 0,C 180,E1 -4181.903,E2 -4181.903} C_VEL
LIN {X 0,Y 532.104,Z 450.211,A -85,B 0,C 180,E1 -4182.721,E2 -4182.721} C_VEL
LIN {X 0,Y 531.056,Z 450.338,A -85,B 0,C 180,E1 -4183.352,E2 -4183.352} C_VEL
LIN {X 0,Y 530.968,Z 450.347,A -85,B 0,C 180,E1 -4183.565,E2 -4183.565} C_VEL
LIN {X 0,Y 530.969,Z 450.349,A -85,B 0,C 180,E1 -4186.506,E2 -4186.506} C_VEL
LIN {X 0,Y 530.984,Z 450.345,A -85,B 0,C 180,E1 -4189.567,E2 -4189.567} C_VEL
LIN {X 0,Y 530.972,Z 450.347,A -85,B 0,C 180,E1 -4192.577,E2 -4192.577} C_VEL
LIN {X 0,Y 531.001,Z 450.339,A -85,B 0,C 180,E1 -4195.311,E2 -4195.311} C_VEL
LIN {X 0,Y 530.971,Z 450.345,A -85,B 0,C 180,E1 -4198.032,E2 -4198.032} C_VEL
LIN {X 0,Y 530.993,Z 450.343,A -85,B 0,C 180,E1 -4200.874,E2 -4200.874} C_VEL
LIN {X 0,Y 531.002,Z 450.34,A -85,B 0,C 180,E1 -4203.256,E2 -4203.256} C_VEL
LIN {X 0,Y 530.99,Z 450.342,A -85,B 0,C 180,E1 -4205.961,E2 -4205.961} C_VEL
LIN {X 0,Y 531.003,Z 450.339,A -85,B 0,C 180,E1 -4209.062,E2 -4209.062} C_VEL
LIN {X 0,Y 530.991,Z 450.345,A -85,B 0,C 180,E1 -4211.479,E2 -4211.479} C_VEL
LIN {X 0,Y 531,Z 450.344,A -85,B 0,C 180,E1 -4214.65,E2 -4214.65} C_VEL
LIN {X 0,Y 531.046,Z 450.339,A -85,B 0,C 180,E1 -4217.775,E2 -4217.775} C_VEL
LIN {X 0,Y 531.028,Z 450.341,A -85,B 0,C 180,E1 -4220.862,E2 -4220.862} C_VEL
LIN {X 0,Y 531.021,Z 450.337,A -85,B 0,C 180,E1 -4223.159,E2 -4223.159} C_VEL
LIN {X 0,Y 531.121,Z 450.325,A -85,B 0,C 180,E1 -4224.685,E2 -4224.685} C_VEL
LIN {X 0,Y 531.145,Z 450.323,A -85,B 0,C 180,E1 -4227.725,E2 -4227.725} C_VEL
LIN {X 0,Y 531.157,Z 450.32,A -85,B 0,C 180,E1 -4230.758,E2 -4230.758} C_VEL
LIN {X 0,Y 531.108,Z 450.329,A -85,B 0,C 180,E1 -4233.034,E2 -4233.034} C_VEL
LIN {X 0,Y 531.09,Z 450.331,A -85,B 0,C 180,E1 -4236.077,E2 -4236.077} C_VEL
LIN {X 0,Y 531.029,Z 450.337,A -85,B 0,C 180,E1 -4239.138,E2 -4239.138} C_VEL
LIN {X 0,Y 531.047,Z 450.336,A -85,B 0,C 180,E1 -4242.225,E2 -4242.225} C_VEL
LIN {X 0,Y 531,Z 450.34,A -85,B 0,C 180,E1 -4245.35,E2 -4245.35} C_VEL
LIN {X 0,Y 530.993,Z 450.342,A -85,B 0,C 180,E1 -4248.521,E2 -4248.521} C_VEL
LIN {X 0,Y 531.004,Z 450.341,A -85,B 0,C 180,E1 -4250.938,E2 -4250.938} C_VEL
LIN {X 0,Y 530.977,Z 450.343,A -85,B 0,C 180,E1 -4254.225,E2 -4254.225} C_VEL
LIN {X 0,Y 531.007,Z 450.343,A -85,B 0,C 180,E1 -4256.744,E2 -4256.744} C_VEL
LIN {X 0,Y 530.987,Z 450.342,A -85,B 0,C 180,E1 -4259.323,E2 -4259.323} C_VEL
LIN {X 0,Y 530.97,Z 450.344,A -85,B 0,C 180,E1 -4262.1,E2 -4262.1} C_VEL
LIN {X 0,Y 530.976,Z 450.346,A -85,B 0,C 180,E1 -4264.851,E2 -4264.851} C_VEL
LIN {X 0,Y 530.97,Z 450.347,A -85,B 0,C 180,E1 -4267.508,E2 -4267.508} C_VEL
LIN {X 0,Y 530.987,Z 450.344,A -85,B 0,C 180,E1 -4270.433,E2 -4270.433} C_VEL
LIN {X 0,Y 530.965,Z 450.344,A -85,B 0,C 180,E1 -4273.281,E2 -4273.281} C_VEL
LIN {X 0,Y 530.986,Z 450.346,A -85,B 0,C 180,E1 -4275.621,E2 -4275.621} C_VEL
LIN {X 0,Y 531.002,Z 450.344,A -85,B 0,C 180,E1 -4278.565,E2 -4278.565} C_VEL
LIN {X 0,Y 530.96,Z 450.348,A -85,B 0,C 180,E1 -4281.529,E2 -4281.529} C_VEL
LIN {X 0,Y 530.914,Z 450.352,A -85,B 0,C 180,E1 -4284.376,E2 -4284.376} C_VEL
LIN {X 0,Y 530.732,Z 450.378,A -85,B 0,C 180,E1 -4286.538,E2 -4286.538} C_VEL
LIN {X 0,Y 530.653,Z 450.389,A -85,B 0,C 180,E1 -4287.111,E2 -4287.111} C_VEL
LIN {X 0,Y 530.609,Z 451.984,A -85,B 0,C 180,E1 -4288.898,E2 -4288.898} C_VEL
LIN {X 0,Y 530.571,Z 454.883,A -85,B 0,C 180,E1 -4291.519,E2 -4291.519} C_VEL
LIN {X 0,Y 530.589,Z 457.898,A -85,B 0,C 180,E1 -4294.251,E2 -4294.251} C_VEL
LIN {X 0,Y 530.503,Z 460.532,A -85,B 0,C 180,E1 -4296.582,E2 -4296.582} C_VEL
LIN {X 0,Y 530.467,Z 463.289,A -85,B 0,C 180,E1 -4299.04,E2 -4299.04} C_VEL
LIN {X 0,Y 530.461,Z 466.039,A -85,B 0,C 180,E1 -4301.459,E2 -4301.459} C_VEL
LIN {X 0,Y 530.436,Z 468.708,A -85,B 0,C 180,E1 -4303.845,E2 -4303.845} C_VEL
LIN {X 0,Y 530.43,Z 471.82,A -85,B 0,C 180,E1 -4306.568,E2 -4306.568} C_VEL
LIN {X 0,Y 532.244,Z 482.813,A -85,B 0,C 180,E1 -4306.906,E2 -4306.906} C_VEL
LIN {X 0,Y 532.052,Z 495.321,A -85,B 0,C 180,E1 -4307.363,E2 -4307.363} C_VEL
LIN {X 0,Y 531.796,Z 507.184,A -85,B 0,C 180,E1 -4307.948,E2 -4307.948} C_VEL
LIN {X 0,Y 531.588,Z 518.298,A -85,B 0,C 180,E1 -4308.658,E2 -4308.658} C_VEL
LIN {X 0,Y 531.288,Z 529.033,A -85,B 0,C 180,E1 -4309.52,E2 -4309.52} C_VEL
LIN {X 0,Y 531.071,Z 538.695,A -85,B 0,C 180,E1 -4310.478,E2 -4310.478} C_VEL
LIN {X 0,Y 530.891,Z 546.612,A -85,B 0,C 180,E1 -4311.435,E2 -4311.435} C_VEL
LIN {X 0,Y 530.691,Z 554.358,A -85,B 0,C 180,E1 -4312.581,E2 -4312.581} C_VEL
LIN {X 0,Y 530.607,Z 561.464,A -85,B 0,C 180,E1 -4313.917,E2 -4313.917} C_VEL
LIN {X 0,Y 530.459,Z 566.203,A -85,B 0,C 180,E1 -4315.06,E2 -4315.06} C_VEL
LIN {X 0,Y 530.516,Z 569.834,A -85,B 0,C 180,E1 -4316.202,E2 -4316.202} C_VEL
LIN {X 0,Y 530.457,Z 571.71,A -85,B 0,C 180,E1 -4316.962,E2 -4316.962} C_VEL
LIN {X 0,Y 530.411,Z 573.129,A -85,B 0,C 180,E1 -4317.722,E2 -4317.722} C_VEL
LIN {X 0,Y 530.345,Z 574.758,A -85,B 0,C 180,E1 -4319.241,E2 -4319.241} C_VEL
LIN {X 0,Y 530.343,Z 574.997,A -85,B 0,C 180,E1 -4320,E2 -4320} C_VEL
LIN {X 0,Y 530.344,Z 574.814,A -85,B 0,C 180,E1 -4320.759,E2 -4320.759} C_VEL
LIN {X 0,Y 530.41,Z 573.26,A -85,B 0,C 180,E1 -4322.278,E2 -4322.278} C_VEL
LIN {X 0,Y 530.458,Z 571.899,A -85,B 0,C 180,E1 -4323.038,E2 -4323.038} C_VEL
LIN {X 0,Y 530.523,Z 569.021,A -85,B 0,C 180,E1 -4324.178,E2 -4324.178} C_VEL
LIN {X 0,Y 530.524,Z 565.118,A -85,B 0,C 180,E1 -4325.321,E2 -4325.321} C_VEL
LIN {X 0,Y 530.594,Z 559.528,A -85,B 0,C 180,E1 -4326.577,E2 -4326.577} C_VEL
LIN {X 0,Y 530.758,Z 552.525,A -85,B 0,C 180,E1 -4327.8,E2 -4327.8} C_VEL
LIN {X 0,Y 530.903,Z 544.341,A -85,B 0,C 180,E1 -4328.948,E2 -4328.948} C_VEL
LIN {X 0,Y 531.106,Z 535.969,A -85,B 0,C 180,E1 -4329.906,E2 -4329.906} C_VEL
LIN {X 0,Y 531.399,Z 525.639,A -85,B 0,C 180,E1 -4330.863,E2 -4330.863} C_VEL
LIN {X 0,Y 531.694,Z 513.925,A -85,B 0,C 180,E1 -4331.73,E2 -4331.73} C_VEL
LIN {X 0,Y 531.913,Z 502.419,A -85,B 0,C 180,E1 -4332.398,E2 -4332.398} C_VEL
LIN {X 0,Y 532.137,Z 490.404,A -85,B 0,C 180,E1 -4332.926,E2 -4332.926} C_VEL
LIN {X 0,Y 532.131,Z 481.436,A -85,B 0,C 180,E1 -4333.23,E2 -4333.23} C_VEL
LIN {X 0,Y 530.438,Z 471.988,A -85,B 0,C 180,E1 -4333.504,E2 -4333.504} C_VEL
LIN {X 0,Y 530.464,Z 469.139,A -85,B 0,C 180,E1 -4336.154,E2 -4336.154} C_VEL
LIN {X 0,Y 530.477,Z 466.671,A -85,B 0,C 180,E1 -4338.54,E2 -4338.54} C_VEL
LIN {X 0,Y 530.578,Z 464.221,A -85,B 0,C 180,E1 -4340.955,E2 -4340.955} C_VEL
LIN {X 0,Y 530.641,Z 460.879,A -85,B 0,C 180,E1 -4344.241,E2 -4344.241} C_VEL
LIN {X 0,Y 530.717,Z 458.411,A -85,B 0,C 180,E1 -4346.759,E2 -4346.759} C_VEL
LIN {X 0,Y 530.765,Z 455.921,A -85,B 0,C 180,E1 -4349.336,E2 -4349.336} C_VEL
LIN {X 0,Y 530.867,Z 453.415,A -85,B 0,C 180,E1 -4352.083,E2 -4352.083} C_VEL
LIN {X 0,Y 530.933,Z 450.968,A -85,B 0,C 180,E1 -4354.845,E2 -4354.845} C_VEL
LIN {X 0,Y 530.896,Z 450.358,A -85,B 0,C 180,E1 -4355.625,E2 -4355.625} C_VEL
LIN {X 0,Y 530.961,Z 450.349,A -85,B 0,C 180,E1 -4358.47,E2 -4358.47} C_VEL
LIN {X 0,Y 531.001,Z 450.345,A -85,B 0,C 180,E1 -4361.435,E2 -4361.435} C_VEL
LIN {X 0,Y 530.992,Z 450.345,A -85,B 0,C 180,E1 -4364.547,E2 -4364.547} C_VEL
LIN {X 0,Y 530.987,Z 450.347,A -85,B 0,C 180,E1 -4367.834,E2 -4367.834} C_VEL
LIN {X 0,Y 531.046,Z 450.481,A -85,B 0,C 180,E1 -4370.459,E2 -4370.459} C_VEL
LIN {X 0,Y 531.661,Z 453.924,A -85,B 0,C 180,E1 -4372.55,E2 -4372.55} C_VEL
LIN {X 0,Y 532.132,Z 457.842,A -85,B 0,C 180,E1 -4374.47,E2 -4374.47} C_VEL
LIN {X 0,Y 531.783,Z 463.52,A -85,B 0,C 180,E1 -4376.771,E2 -4376.771} C_VEL
LIN {X 0,Y 531.517,Z 472.015,A -85,B 0,C 180,E1 -4379.837,E2 -4379.837} C_VEL
LIN {X 0,Y 531.312,Z 481.165,A -85,B 0,C 180,E1 -4382.848,E2 -4382.848} C_VEL
LIN {X 0,Y 531.089,Z 491.211,A -85,B 0,C 180,E1 -4385.936,E2 -4385.936} C_VEL
LIN {X 0,Y 530.975,Z 500.298,A -85,B 0,C 180,E1 -4388.654,E2 -4388.654} C_VEL
LIN {X 0,Y 530.882,Z 510.115,A -85,B 0,C 180,E1 -4391.475,E2 -4391.475} C_VEL
LIN {X 0,Y 530.787,Z 521.234,A -85,B 0,C 180,E1 -4394.644,E2 -4394.644} C_VEL
LIN {X 0,Y 530.709,Z 527.53,A -85,B 0,C 180,E1 -4396.454,E2 -4396.454} C_VEL
LIN {X 0,Y 532.331,Z 538.345,A -85,B 0,C 180,E1 -4396.739,E2 -4396.739} C_VEL
LIN {X 0,Y 532.122,Z 551.77,A -85,B 0,C 180,E1 -4397.17,E2 -4397.17} C_VEL
LIN {X 0,Y 531.932,Z 563.404,A -85,B 0,C 180,E1 -4397.699,E2 -4397.699} C_VEL
LIN {X 0,Y 531.637,Z 575.805,A -85,B 0,C 180,E1 -4398.441,E2 -4398.441} C_VEL
LIN {X 0,Y 531.384,Z 586.264,A -85,B 0,C 180,E1 -4399.233,E2 -4399.233} C_VEL
LIN {X 0,Y 531.113,Z 595.538,A -85,B 0,C 180,E1 -4400.094,E2 -4400.094} C_VEL
LIN {X 0,Y 530.931,Z 603.991,A -85,B 0,C 180,E1 -4401.052,E2 -4401.052} C_VEL
LIN {X 0,Y 530.758,Z 612.234,A -85,B 0,C 180,E1 -4402.199,E2 -4402.199} C_VEL
LIN {X 0,Y 530.598,Z 619.268,A -85,B 0,C 180,E1 -4403.419,E2 -4403.419} C_VEL
LIN {X 0,Y 530.525,Z 624.949,A -85,B 0,C 180,E1 -4404.679,E2 -4404.679} C_VEL
LIN {X 0,Y 530.522,Z 628.894,A -85,B 0,C 180,E1 -4405.822,E2 -4405.822} C_VEL
LIN {X 0,Y 530.457,Z 631.807,A -85,B 0,C 180,E1 -4406.962,E2 -4406.962} C_VEL
LIN {X 0,Y 530.41,Z 633.194,A -85,B 0,C 180,E1 -4407.722,E2 -4407.722} C_VEL
LIN {X 0,Y 530.344,Z 634.786,A -85,B 0,C 180,E1 -4409.241,E2 -4409.241} C_VEL
LIN {X 0,Y 530.342,Z 635,A -85,B 0,C 180,E1 -4410,E2 -4410} C_VEL
LIN {X 0,Y 530.361,Z 634.184,A -85,B 0,C 180,E1 -4411.519,E2 -4411.519} C_VEL
LIN {X 0,Y 530.41,Z 633.197,A -85,B 0,C 180,E1 -4412.278,E2 -4412.278} C_VEL
LIN {X 0,Y 530.457,Z 631.81,A -85,B 0,C 180,E1 -4413.038,E2 -4413.038} C_VEL
LIN {X 0,Y 530.522,Z 628.895,A -85,B 0,C 180,E1 -4414.178,E2 -4414.178} C_VEL
LIN {X 0,Y 530.525,Z 624.948,A -85,B 0,C 180,E1 -4415.321,E2 -4415.321} C_VEL
LIN {X 0,Y 530.599,Z 619.263,A -85,B 0,C 180,E1 -4416.582,E2 -4416.582} C_VEL
LIN {X 0,Y 530.758,Z 612.236,A -85,B 0,C 180,E1 -4417.8,E2 -4417.8} C_VEL
LIN {X 0,Y 530.931,Z 603.992,A -85,B 0,C 180,E1 -4418.948,E2 -4418.948} C_VEL
LIN {X 0,Y 531.113,Z 595.54,A -85,B 0,C 180,E1 -4419.905,E2 -4419.905} C_VEL
LIN {X 0,Y 531.407,Z 585.092,A -85,B 0,C 180,E1 -4420.863,E2 -4420.863} C_VEL
LIN {X 0,Y 531.675,Z 574.172,A -85,B 0,C 180,E1 -4421.669,E2 -4421.669} C_VEL
LIN {X 0,Y 531.934,Z 563.405,A -85,B 0,C 180,E1 -4422.301,E2 -4422.301} C_VEL
LIN {X 0,Y 532.118,Z 551.765,A -85,B 0,C 180,E1 -4422.83,E2 -4422.83} C_VEL
LIN {X 0,Y 532.301,Z 538.345,A -85,B 0,C 180,E1 -4423.262,E2 -4423.262} C_VEL
LIN {X 0,Y 530.709,Z 527.53,A -85,B 0,C 180,E1 -4423.546,E2 -4423.546} C_VEL
LIN {X 0,Y 530.817,Z 518.586,A -85,B 0,C 180,E1 -4426.143,E2 -4426.143} C_VEL
LIN {X 0,Y 530.915,Z 509.055,A -85,B 0,C 180,E1 -4428.924,E2 -4428.924} C_VEL
LIN {X 0,Y 531.055,Z 499.585,A -85,B 0,C 180,E1 -4431.75,E2 -4431.75} C_VEL
LIN {X 0,Y 531.23,Z 490.288,A -85,B 0,C 180,E1 -4434.629,E2 -4434.629} C_VEL
LIN {X 0,Y 531.436,Z 480.853,A -85,B 0,C 180,E1 -4437.619,E2 -4437.619} C_VEL
LIN {X 0,Y 531.715,Z 471.209,A -85,B 0,C 180,E1 -4440.779,E2 -4440.779} C_VEL
LIN {X 0,Y 531.977,Z 462.665,A -85,B 0,C 180,E1 -4443.702,E2 -4443.702} C_VEL
LIN {X 0,Y 532.078,Z 457.509,A -85,B 0,C 180,E1 -4445.533,E2 -4445.533} C_VEL
LIN {X 0,Y 531.348,Z 452.359,A -85,B 0,C 180,E1 -4447.476,E2 -4447.476} C_VEL
LIN {X 0,Y 530.985,Z 450.347,A -85,B 0,C 180,E1 -4448.347,E2 -4448.347} C_VEL
LIN {X 0,Y 530.998,Z 450.346,A -85,B 0,C 180,E1 -4451.435,E2 -4451.435} C_VEL
LIN {X 0,Y 530.991,Z 450.346,A -85,B 0,C 180,E1 -4454.547,E2 -4454.547} C_VEL
LIN {X 0,Y 530.989,Z 450.345,A -85,B 0,C 180,E1 -4457.834,E2 -4457.834} C_VEL
LIN {X 0,Y 530.987,Z 450.345,A -85,B 0,C 180,E1 -4460.557,E2 -4460.557} C_VEL
LIN {X 0,Y 530.957,Z 450.347,A -85,B 0,C 180,E1 -4463.442,E2 -4463.442} C_VEL
LIN {X 0,Y 531,Z 450.341,A -85,B 0,C 180,E1 -4466.494,E2 -4466.494} C_VEL
LIN {X 0,Y 530.976,Z 450.343,A -85,B 0,C 180,E1 -4469.355,E2 -4469.355} C_VEL
LIN {X 0,Y 531.017,Z 450.338,A -85,B 0,C 180,E1 -4472.467,E2 -4472.467} C_VEL
LIN {X 0,Y 530.997,Z 450.344,A -85,B 0,C 180,E1 -4474.942,E2 -4474.942} C_VEL
LIN {X 0,Y 530.974,Z 450.346,A -85,B 0,C 180,E1 -4478.247,E2 -4478.247} C_VEL
LIN {X 0,Y 530.998,Z 450.342,A -85,B 0,C 180,E1 -4480.677,E2 -4480.677} C_VEL
LIN {X 0,Y 530.988,Z 450.342,A -85,B 0,C 180,E1 -4483.071,E2 -4483.071} C_VEL
LIN {X 0,Y 531.022,Z 450.34,A -85,B 0,C 180,E1 -4485.436,E2 -4485.436} C_VEL
LIN {X 0,Y 531.04,Z 450.338,A -85,B 0,C 180,E1 -4488.55,E2 -4488.55} C_VEL
LIN {X 0,Y 531.057,Z 450.335,A -85,B 0,C 180,E1 -4491.63,E2 -4491.63} C_VEL
LIN {X 0,Y 531.124,Z 450.327,A -85,B 0,C 180,E1 -4494.685,E2 -4494.685} C_VEL
LIN {X 0,Y 531.14,Z 450.323,A -85,B 0,C 180,E1 -4497.725,E2 -4497.725} C_VEL
LIN {X 0,Y 531.157,Z 450.321,A -85,B 0,C 180,E1 -4500.758,E2 -4500.758} C_VEL
LIN {X 0,Y 531.108,Z 450.33,A -85,B 0,C 180,E1 -4503.034,E2 -4503.034} C_VEL
LIN {X 0,Y 531.086,Z 450.335,A -85,B 0,C 180,E1 -4506.077,E2 -4506.077} C_VEL
LIN {X 0,Y 531.033,Z 450.34,A -85,B 0,C 180,E1 -4509.138,E2 -4509.138} C_VEL
LIN {X 0,Y 531.043,Z 450.339,A -85,B 0,C 180,E1 -4512.225,E2 -4512.225} C_VEL
LIN {X 0,Y 530.999,Z 450.344,A -85,B 0,C 180,E1 -4515.35,E2 -4515.35} C_VEL
LIN {X 0,Y 530.993,Z 450.346,A -85,B 0,C 180,E1 -4518.521,E2 -4518.521} C_VEL
LIN {X 0,Y 531.003,Z 450.34,A -85,B 0,C 180,E1 -4520.938,E2 -4520.938} C_VEL
LIN {X 0,Y 530.975,Z 450.344,A -85,B 0,C 180,E1 -4524.225,E2 -4524.225} C_VEL
LIN {X 0,Y 531.008,Z 450.34,A -85,B 0,C 180,E1 -4526.744,E2 -4526.744} C_VEL
LIN {X 0,Y 530.985,Z 450.346,A -85,B 0,C 180,E1 -4529.323,E2 -4529.323} C_VEL
LIN {X 0,Y 530.974,Z 450.345,A -85,B 0,C 180,E1 -4532.101,E2 -4532.101} C_VEL
LIN {X 0,Y 530.988,Z 450.342,A -85,B 0,C 180,E1 -4534.854,E2 -4534.854} C_VEL
LIN {X 0,Y 530.97,Z 450.347,A -85,B 0,C 180,E1 -4537.508,E2 -4537.508} C_VEL
LIN {X 0,Y 530.985,Z 450.346,A -85,B 0,C 180,E1 -4540.433,E2 -4540.433} C_VEL
LIN {X 0,Y 530.971,Z 450.348,A -85,B 0,C 180,E1 -4543.495,E2 -4543.495} C_VEL
LIN {X 0,Y 530.968,Z 450.347,A -85,B 0,C 180,E1 -4543.565,E2 -4543.565} C_VEL
LIN {X 0,Y 530.294,Z 450.429,A -85,B 0,C 180,E1 -4544.199,E2 -4544.199} C_VEL
LIN {X 0,Y 527.447,Z 450.786,A -85,B 0,C 180,E1 -4545.228,E2 -4545.228} C_VEL
LIN {X 0,Y 525.043,Z 451.087,A -85,B 0,C 180,E1 -4546.056,E2 -4546.056} C_VEL
LIN {X 0,Y 524.008,Z 451.214,A -85,B 0,C 180,E1 -4546.696,E2 -4546.696} C_VEL
LIN {X 0,Y 523.923,Z 451.223,A -85,B 0,C 180,E1 -4546.912,E2 -4546.912} C_VEL
LIN {X 0,Y 523.952,Z 451.221,A -85,B 0,C 180,E1 -4549.921,E2 -4549.921} C_VEL
LIN {X 0,Y 523.914,Z 451.226,A -85,B 0,C 180,E1 -4552.868,E2 -4552.868} C_VEL
LIN {X 0,Y 523.946,Z 451.221,A -85,B 0,C 180,E1 -4555.711,E2 -4555.711} C_VEL
LIN {X 0,Y 523.925,Z 451.222,A -85,B 0,C 180,E1 -4558.456,E2 -4558.456} C_VEL
LIN {X 0,Y 523.942,Z 451.219,A -85,B 0,C 180,E1 -4561.125,E2 -4561.125} C_VEL
LIN {X 0,Y 523.988,Z 451.217,A -85,B 0,C 180,E1 -4563.981,E2 -4563.981} C_VEL
LIN {X 0,Y 523.931,Z 451.222,A -85,B 0,C 180,E1 -4566.271,E2 -4566.271} C_VEL
LIN {X 0,Y 523.95,Z 451.219,A -85,B 0,C 180,E1 -4568.767,E2 -4568.767} C_VEL
LIN {X 0,Y 523.953,Z 451.22,A -85,B 0,C 180,E1 -4571.221,E2 -4571.221} C_VEL
LIN {X 0,Y 523.936,Z 451.221,A -85,B 0,C 180,E1 -4573.639,E2 -4573.639} C_VEL
LIN {X 0,Y 523.945,Z 451.222,A -85,B 0,C 180,E1 -4576.028,E2 -4576.028} C_VEL
LIN {X 0,Y 524.018,Z 451.21,A -85,B 0,C 180,E1 -4578.394,E2 -4578.394} C_VEL
LIN {X 0,Y 524.007,Z 451.212,A -85,B 0,C 180,E1 -4581.516,E2 -4581.516} C_VEL
LIN {X 0,Y 524.081,Z 451.202,A -85,B 0,C 180,E1 -4584.614,E2 -4584.614} C_VEL
LIN {X 0,Y 524.117,Z 451.198,A -85,B 0,C 180,E1 -4587.695,E2 -4587.695} C_VEL
LIN {X 0,Y 524.127,Z 451.196,A -85,B 0,C 180,E1 -4590.768,E2 -4590.768} C_VEL
LIN {X 0,Y 524.075,Z 451.205,A -85,B 0,C 180,E1 -4593.075,E2 -4593.075} C_VEL
LIN {X 0,Y 524.052,Z 451.208,A -85,B 0,C 180,E1 -4596.159,E2 -4596.159} C_VEL
LIN {X 0,Y 523.999,Z 451.213,A -85,B 0,C 180,E1 -4599.262,E2 -4599.262} C_VEL
LIN {X 0,Y 524.009,Z 451.212,A -85,B 0,C 180,E1 -4601.74,E2 -4601.74} C_VEL
LIN {X 0,Y 523.999,Z 451.211,A -85,B 0,C 180,E1 -4605.052,E2 -4605.052} C_VEL
LIN {X 0,Y 523.969,Z 451.217,A -85,B 0,C 180,E1 -4607.969,E2 -4607.969} C_VEL
LIN {X 0,Y 523.977,Z 451.22,A -85,B 0,C 180,E1 -4610.41,E2 -4610.41} C_VEL
LIN {X 0,Y 523.917,Z 451.221,A -85,B 0,C 180,E1 -4612.893,E2 -4612.893} C_VEL
LIN {X 0,Y 523.959,Z 451.221,A -85,B 0,C 180,E1 -4615.419,E2 -4615.419} C_VEL
LIN {X 0,Y 523.973,Z 451.218,A -85,B 0,C 180,E1 -4617.999,E2 -4617.999} C_VEL
LIN {X 0,Y 523.95,Z 451.218,A -85,B 0,C 180,E1 -4620.855,E2 -4620.855} C_VEL
LIN {X 0,Y 523.964,Z 451.217,A -85,B 0,C 180,E1 -4623.734,E2 -4623.734} C_VEL
LIN {X 0,Y 523.908,Z 451.225,A -85,B 0,C 180,E1 -4626.401,E2 -4626.401} C_VEL
LIN {X 0,Y 523.926,Z 451.224,A -85,B 0,C 180,E1 -4629.085,E2 -4629.085} C_VEL
LIN {X 0,Y 523.959,Z 451.221,A -85,B 0,C 180,E1 -4632.119,E2 -4632.119} C_VEL
LIN {X 0,Y 523.95,Z 451.221,A -85,B 0,C 180,E1 -4635.31,E2 -4635.31} C_VEL
LIN {X 0,Y 523.964,Z 451.22,A -85,B 0,C 180,E1 -4638.689,E2 -4638.689} C_VEL
LIN {X 0,Y 523.921,Z 451.222,A -85,B 0,C 180,E1 -4641.081,E2 -4641.081} C_VEL
LIN {X 0,Y 523.875,Z 451.229,A -85,B 0,C 180,E1 -4643.823,E2 -4643.823} C_VEL
LIN {X 0,Y 523.733,Z 451.25,A -85,B 0,C 180,E1 -4646.303,E2 -4646.303} C_VEL
LIN {X 0,Y 523.555,Z 451.368,A -85,B 0,C 180,E1 -4647.746,E2 -4647.746} C_VEL
LIN {X 0,Y 523.521,Z 454.056,A -85,B 0,C 180,E1 -4650.217,E2 -4650.217} C_VEL
LIN {X 0,Y 523.514,Z 456.949,A -85,B 0,C 180,E1 -4652.842,E2 -4652.842} C_VEL
LIN {X 0,Y 523.435,Z 459.794,A -85,B 0,C 180,E1 -4655.403,E2 -4655.403} C_VEL
LIN {X 0,Y 523.442,Z 462.595,A -85,B 0,C 180,E1 -4657.917,E2 -4657.917} C_VEL
LIN {X 0,Y 523.412,Z 465.366,A -85,B 0,C 180,E1 -4660.386,E2 -4660.386} C_VEL
LIN {X 0,Y 523.382,Z 468.1,A -85,B 0,C 180,E1 -4662.817,E2 -4662.817} C_VEL
LIN {X 0,Y 523.377,Z 471.975,A -85,B 0,C 180,E1 -4666.211,E2 -4666.211} C_VEL
LIN {X 0,Y 523.395,Z 472.431,A -85,B 0,C 180,E1 -4666.409,E2 -4666.409} C_VEL
LIN {X 0,Y 525.327,Z 483.716,A -85,B 0,C 180,E1 -4666.755,E2 -4666.755} C_VEL
LIN {X 0,Y 525.108,Z 496.611,A -85,B 0,C 180,E1 -4667.242,E2 -4667.242} C_VEL
LIN {X 0,Y 524.842,Z 508.137,A -85,B 0,C 180,E1 -4667.83,E2 -4667.83} C_VEL
LIN {X 0,Y 524.571,Z 519.767,A -85,B 0,C 180,E1 -4668.602,E2 -4668.602} C_VEL
LIN {X 0,Y 524.279,Z 530.259,A -85,B 0,C 180,E1 -4669.476,E2 -4669.476} C_VEL
LIN {X 0,Y 524.06,Z 538.826,A -85,B 0,C 180,E1 -4670.35,E2 -4670.35} C_VEL
LIN {X 0,Y 523.859,Z 546.707,A -85,B 0,C 180,E1 -4671.319,E2 -4671.319} C_VEL
LIN {X 0,Y 523.638,Z 554.41,A -85,B 0,C 180,E1 -4672.481,E2 -4672.481} C_VEL
LIN {X 0,Y 523.519,Z 561.467,A -85,B 0,C 180,E1 -4673.835,E2 -4673.835} C_VEL
LIN {X 0,Y 523.384,Z 566.205,A -85,B 0,C 180,E1 -4674.993,E2 -4674.993} C_VEL
LIN {X 0,Y 523.444,Z 569.835,A -85,B 0,C 180,E1 -4676.151,E2 -4676.151} C_VEL
LIN {X 0,Y 523.368,Z 571.712,A -85,B 0,C 180,E1 -4676.921,E2 -4676.921} C_VEL
LIN {X 0,Y 523.334,Z 573.13,A -85,B 0,C 180,E1 -4677.691,E2 -4677.691} C_VEL
LIN {X 0,Y 523.251,Z 574.758,A -85,B 0,C 180,E1 -4679.23,E2 -4679.23} C_VEL
LIN {X 0,Y 523.247,Z 574.997,A -85,B 0,C 180,E1 -4680,E2 -4680} C_VEL
LIN {X 0,Y 523.25,Z 574.813,A -85,B 0,C 180,E1 -4680.769,E2 -4680.769} C_VEL
LIN {X 0,Y 523.334,Z 573.258,A -85,B 0,C 180,E1 -4682.309,E2 -4682.309} C_VEL
LIN {X 0,Y 523.368,Z 571.897,A -85,B 0,C 180,E1 -4683.079,E2 -4683.079} C_VEL
LIN {X 0,Y 523.441,Z 569.019,A -85,B 0,C 180,E1 -4684.235,E2 -4684.235} C_VEL
LIN {X 0,Y 523.463,Z 565.116,A -85,B 0,C 180,E1 -4685.393,E2 -4685.393} C_VEL
LIN {X 0,Y 523.518,Z 559.983,A -85,B 0,C 180,E1 -4686.575,E2 -4686.575} C_VEL
LIN {X 0,Y 523.665,Z 553.814,A -85,B 0,C 180,E1 -4687.713,E2 -4687.713} C_VEL
LIN {X 0,Y 523.856,Z 545.945,A -85,B 0,C 180,E1 -4688.875,E2 -4688.875} C_VEL
LIN {X 0,Y 524.099,Z 536.144,A -85,B 0,C 180,E1 -4690.039,E2 -4690.039} C_VEL
LIN {X 0,Y 524.423,Z 525.839,A -85,B 0,C 180,E1 -4691.009,E2 -4691.009} C_VEL
LIN {X 0,Y 524.717,Z 515.714,A -85,B 0,C 180,E1 -4691.78,E2 -4691.78} C_VEL
LIN {X 0,Y 524.957,Z 504.444,A -85,B 0,C 180,E1 -4692.467,E2 -4692.467} C_VEL
LIN {X 0,Y 525.176,Z 493.108,A -85,B 0,C 180,E1 -4693.002,E2 -4693.002} C_VEL
LIN {X 0,Y 525.182,Z 482.283,A -85,B 0,C 180,E1 -4693.386,E2 -4693.386} C_VEL
LIN {X 0,Y 523.373,Z 472.476,A -85,B 0,C 180,E1 -4693.69,E2 -4693.69} C_VEL
LIN {X 0,Y 523.399,Z 469.605,A -85,B 0,C 180,E1 -4696.378,E2 -4696.378} C_VEL
LIN {X 0,Y 523.488,Z 466.332,A -85,B 0,C 180,E1 -4699.611,E2 -4699.611} C_VEL
LIN {X 0,Y 523.519,Z 463.764,A -85,B 0,C 180,E1 -4702.135,E2 -4702.135} C_VEL
LIN {X 0,Y 523.599,Z 461.348,A -85,B 0,C 180,E1 -4704.588,E2 -4704.588} C_VEL
LIN {X 0,Y 523.711,Z 458.395,A -85,B 0,C 180,E1 -4707.662,E2 -4707.662} C_VEL
LIN {X 0,Y 523.776,Z 455.463,A -85,B 0,C 180,E1 -4710.823,E2 -4710.823} C_VEL
LIN {X 0,Y 523.901,Z 452.955,A -85,B 0,C 180,E1 -4713.724,E2 -4713.724} C_VEL
LIN {X 0,Y 523.888,Z 451.707,A -85,B 0,C 180,E1 -4715.229,E2 -4715.229} C_VEL
LIN {X 0,Y 523.886,Z 451.232,A -85,B 0,C 180,E1 -4716.398,E2 -4716.398} C_VEL
LIN {X 0,Y 523.924,Z 451.227,A -85,B 0,C 180,E1 -4719.085,E2 -4719.085} C_VEL
LIN {X 0,Y 523.959,Z 451.221,A -85,B 0,C 180,E1 -4722.118,E2 -4722.118} C_VEL
LIN {X 0,Y 523.959,Z 451.222,A -85,B 0,C 180,E1 -4725.309,E2 -4725.309} C_VEL
LIN {X 0,Y 523.962,Z 451.221,A -85,B 0,C 180,E1 -4728.689,E2 -4728.689} C_VEL
LIN {X 0,Y 523.982,Z 451.376,A -85,B 0,C 180,E1 -4729.923,E2 -4729.923} C_VEL
LIN {X 0,Y 524.602,Z 454.902,A -85,B 0,C 180,E1 -4732.224,E2 -4732.224} C_VEL
LIN {X 0,Y 525.093,Z 458.13,A -85,B 0,C 180,E1 -4733.92,E2 -4733.92} C_VEL
LIN {X 0,Y 525.016,Z 462.363,A -85,B 0,C 180,E1 -4735.79,E2 -4735.79} C_VEL
LIN {X 0,Y 524.595,Z 469.414,A -85,B 0,C 180,E1 -4738.501,E2 -4738.501} C_VEL
LIN {X 0,Y 524.367,Z 475.372,A -85,B 0,C 180,E1 -4740.597,E2 -4740.597} C_VEL
LIN {X 0,Y 524.191,Z 483.55,A -85,B 0,C 180,E1 -4743.311,E2 -4743.311} C_VEL
LIN {X 0,Y 524.028,Z 493.043,A -85,B 0,C 180,E1 -4746.275,E2 -4746.275} C_VEL
LIN {X 0,Y 523.901,Z 502.643,A -85,B 0,C 180,E1 -4749.176,E2 -4749.176} C_VEL
LIN {X 0,Y 523.753,Z 513.432,A -85,B 0,C 180,E1 -4752.311,E2 -4752.311} C_VEL
LIN {X 0,Y 523.696,Z 523.542,A -85,B 0,C 180,E1 -4755.227,E2 -4755.227} C_VEL
LIN {X 0,Y 523.64,Z 527.368,A -85,B 0,C 180,E1 -4756.292,E2 -4756.292} C_VEL
LIN {X 0,Y 525.397,Z 538.818,A -85,B 0,C 180,E1 -4756.585,E2 -4756.585} C_VEL
LIN {X 0,Y 525.195,Z 551.426,A -85,B 0,C 180,E1 -4756.998,E2 -4756.998} C_VEL
LIN {X 0,Y 524.981,Z 563.183,A -85,B 0,C 180,E1 -4757.533,E2 -4757.533} C_VEL
LIN {X 0,Y 524.696,Z 574.313,A -85,B 0,C 180,E1 -4758.191,E2 -4758.191} C_VEL
LIN {X 0,Y 524.431,Z 585.078,A -85,B 0,C 180,E1 -4758.991,E2 -4758.991} C_VEL
LIN {X 0,Y 524.094,Z 595.538,A -85,B 0,C 180,E1 -4759.96,E2 -4759.96} C_VEL
LIN {X 0,Y 523.896,Z 603.991,A -85,B 0,C 180,E1 -4760.931,E2 -4760.931} C_VEL
LIN {X 0,Y 523.688,Z 612.234,A -85,B 0,C 180,E1 -4762.093,E2 -4762.093} C_VEL
LIN {X 0,Y 523.574,Z 617.867,A -85,B 0,C 180,E1 -4763.061,E2 -4763.061} C_VEL
LIN {X 0,Y 523.544,Z 623.365,A -85,B 0,C 180,E1 -4764.222,E2 -4764.222} C_VEL
LIN {X 0,Y 523.361,Z 627.676,A -85,B 0,C 180,E1 -4765.378,E2 -4765.378} C_VEL
LIN {X 0,Y 523.443,Z 629.957,A -85,B 0,C 180,E1 -4766.151,E2 -4766.151} C_VEL
LIN {X 0,Y 523.367,Z 631.806,A -85,B 0,C 180,E1 -4766.921,E2 -4766.921} C_VEL
LIN {X 0,Y 523.334,Z 633.193,A -85,B 0,C 180,E1 -4767.691,E2 -4767.691} C_VEL
LIN {X 0,Y 523.25,Z 634.785,A -85,B 0,C 180,E1 -4769.23,E2 -4769.23} C_VEL
LIN {X 0,Y 523.246,Z 635,A -85,B 0,C 180,E1 -4770,E2 -4770} C_VEL
LIN {X 0,Y 523.274,Z 634.184,A -85,B 0,C 180,E1 -4771.539,E2 -4771.539} C_VEL
LIN {X 0,Y 523.334,Z 633.196,A -85,B 0,C 180,E1 -4772.309,E2 -4772.309} C_VEL
LIN {X 0,Y 523.367,Z 631.81,A -85,B 0,C 180,E1 -4773.079,E2 -4773.079} C_VEL
LIN {X 0,Y 523.441,Z 628.895,A -85,B 0,C 180,E1 -4774.235,E2 -4774.235} C_VEL
LIN {X 0,Y 523.464,Z 624.948,A -85,B 0,C 180,E1 -4775.393,E2 -4775.393} C_VEL
LIN {X 0,Y 523.523,Z 619.727,A -85,B 0,C 180,E1 -4776.581,E2 -4776.581} C_VEL
LIN {X 0,Y 523.665,Z 613.466,A -85,B 0,C 180,E1 -4777.713,E2 -4777.713} C_VEL
LIN {X 0,Y 523.857,Z 605.477,A -85,B 0,C 180,E1 -4778.875,E2 -4778.875} C_VEL
LIN {X 0,Y 524.085,Z 597.333,A -85,B 0,C 180,E1 -4779.845,E2 -4779.845} C_VEL
LIN {X 0,Y 524.362,Z 587.394,A -85,B 0,C 180,E1 -4780.815,E2 -4780.815} C_VEL
LIN {X 0,Y 524.611,Z 577.524,A -85,B 0,C 180,E1 -4781.592,E2 -4781.592} C_VEL
LIN {X 0,Y 524.887,Z 566.063,A -85,B 0,C 180,E1 -4782.312,E2 -4782.312} C_VEL
LIN {X 0,Y 525.135,Z 553.857,A -85,B 0,C 180,E1 -4782.905,E2 -4782.905} C_VEL
LIN {X 0,Y 525.379,Z 540.76,A -85,B 0,C 180,E1 -4783.366,E2 -4783.366} C_VEL
LIN {X 0,Y 524.903,Z 535.239,A -85,B 0,C 180,E1 -4783.523,E2 -4783.523} C_VEL
LIN {X 0,Y 523.642,Z 527.315,A -85,B 0,C 180,E1 -4783.733,E2 -4783.733} C_VEL
LIN {X 0,Y 523.736,Z 518.333,A -85,B 0,C 180,E1 -4786.368,E2 -4786.368} C_VEL
LIN {X 0,Y 523.87,Z 508.799,A -85,B 0,C 180,E1 -4789.189,E2 -4789.189} C_VEL
LIN {X 0,Y 524.023,Z 498.745,A -85,B 0,C 180,E1 -4792.271,E2 -4792.271} C_VEL
LIN {X 0,Y 524.231,Z 490.137,A -85,B 0,C 180,E1 -4794.98,E2 -4794.98} C_VEL
LIN {X 0,Y 524.477,Z 480.881,A -85,B 0,C 180,E1 -4797.969,E2 -4797.969} C_VEL
LIN {X 0,Y 524.745,Z 471.803,A -85,B 0,C 180,E1 -4801,E2 -4801} C_VEL
LIN {X 0,Y 525.022,Z 463.461,A -85,B 0,C 180,E1 -4803.907,E2 -4803.907} C_VEL
LIN {X 0,Y 525.116,Z 458.664,A -85,B 0,C 180,E1 -4805.633,E2 -4805.633} C_VEL
LIN {X 0,Y 524.131,Z 452.313,A -85,B 0,C 180,E1 -4808.083,E2 -4808.083} C_VEL
LIN {X 0,Y 523.939,Z 451.224,A -85,B 0,C 180,E1 -4808.59,E2 -4808.59} C_VEL
LIN {X 0,Y 523.961,Z 451.222,A -85,B 0,C 180,E1 -4811.311,E2 -4811.311} C_VEL
LIN {X 0,Y 523.958,Z 451.221,A -85,B 0,C 180,E1 -4814.691,E2 -4814.691} C_VEL
LIN {X 0,Y 523.958,Z 451.221,A -85,B 0,C 180,E1 -4817.882,E2 -4817.882} C_VEL
LIN {X 0,Y 523.921,Z 451.225,A -85,B 0,C 180,E1 -4820.915,E2 -4820.915} C_VEL
LIN {X 0,Y 523.902,Z 451.228,A -85,B 0,C 180,E1 -4823.825,E2 -4823.825} C_VEL
LIN {X 0,Y 523.943,Z 451.221,A -85,B 0,C 180,E1 -4826.636,E2 -4826.636} C_VEL
LIN {X 0,Y 523.958,Z 451.217,A -85,B 0,C 180,E1 -4829.356,E2 -4829.356} C_VEL
LIN {X 0,Y 523.981,Z 451.215,A -85,B 0,C 180,E1 -4832.281,E2 -4832.281} C_VEL
LIN {X 0,Y 523.949,Z 451.221,A -85,B 0,C 180,E1 -4834.581,E2 -4834.581} C_VEL
LIN {X 0,Y 523.922,Z 451.225,A -85,B 0,C 180,E1 -4837.756,E2 -4837.756} C_VEL
LIN {X 0,Y 523.978,Z 451.215,A -85,B 0,C 180,E1 -4840.408,E2 -4840.408} C_VEL
LIN {X 0,Y 523.969,Z 451.218,A -85,B 0,C 180,E1 -4842.837,E2 -4842.837} C_VEL
LIN {X 0,Y 523.98,Z 451.216,A -85,B 0,C 180,E1 -4845.236,E2 -4845.236} C_VEL
LIN {X 0,Y 524.015,Z 451.211,A -85,B 0,C 180,E1 -4848.394,E2 -4848.394} C_VEL
LIN {X 0,Y 524.006,Z 451.212,A -85,B 0,C 180,E1 -4851.516,E2 -4851.516} C_VEL
LIN {X 0,Y 524.085,Z 451.203,A -85,B 0,C 180,E1 -4854.614,E2 -4854.614} C_VEL
LIN {X 0,Y 524.113,Z 451.198,A -85,B 0,C 180,E1 -4857.695,E2 -4857.695} C_VEL
LIN {X 0,Y 524.127,Z 451.197,A -85,B 0,C 180,E1 -4860.768,E2 -4860.768} C_VEL
LIN {X 0,Y 524.075,Z 451.205,A -85,B 0,C 180,E1 -4863.075,E2 -4863.075} C_VEL
LIN {X 0,Y 524.048,Z 451.21,A -85,B 0,C 180,E1 -4866.159,E2 -4866.159} C_VEL
LIN {X 0,Y 524.001,Z 451.215,A -85,B 0,C 180,E1 -4869.262,E2 -4869.262} C_VEL
LIN {X 0,Y 524.006,Z 451.211,A -85,B 0,C 180,E1 -4871.74,E2 -4871.74} C_VEL
LIN {X 0,Y 523.996,Z 451.215,A -85,B 0,C 180,E1 -4875.053,E2 -4875.053} C_VEL
LIN {X 0,Y 523.967,Z 451.217,A -85,B 0,C 180,E1 -4877.969,E2 -4877.969} C_VEL
LIN {X 0,Y 523.975,Z 451.217,A -85,B 0,C 180,E1 -4880.41,E2 -4880.41} C_VEL
LIN {X 0,Y 523.914,Z 451.226,A -85,B 0,C 180,E1 -4882.894,E2 -4882.894} C_VEL
LIN {X 0,Y 523.956,Z 451.217,A -85,B 0,C 180,E1 -4885.419,E2 -4885.419} C_VEL
LIN {X 0,Y 523.973,Z 451.22,A -85,B 0,C 180,E1 -4887.999,E2 -4887.999} C_VEL
LIN {X 0,Y 523.948,Z 451.223,A -85,B 0,C 180,E1 -4890.855,E2 -4890.855} C_VEL
LIN {X 0,Y 523.964,Z 451.217,A -85,B 0,C 180,E1 -4893.735,E2 -4893.735} C_VEL
LIN {X 0,Y 523.925,Z 451.222,A -85,B 0,C 180,E1 -4896.404,E2 -4896.404} C_VEL
LIN {X 0,Y 523.923,Z 451.223,A -85,B 0,C 180,E1 -4899.085,E2 -4899.085} C_VEL
LIN {X 0,Y 523.96,Z 451.22,A -85,B 0,C 180,E1 -4902.119,E2 -4902.119} C_VEL
LIN {X 0,Y 523.96,Z 451.22,A -85,B 0,C 180,E1 -4905.309,E2 -4905.309} C_VEL
LIN {X 0,Y 523.923,Z 451.223,A -85,B 0,C 180,E1 -4906.912,E2 -4906.912} C_VEL
LIN {X 0,Y 523.255,Z 451.305,A -85,B 0,C 180,E1 -4907.554,E2 -4907.554} C_VEL
LIN {X 0,Y 520.412,Z 451.66,A -85,B 0,C 180,E1 -4908.595,E2 -4908.595} C_VEL
LIN {X 0,Y 518.008,Z 451.961,A -85,B 0,C 180,E1 -4909.434,E2 -4909.434} C_VEL
LIN {X 0,Y 516.972,Z 452.09,A -85,B 0,C 180,E1 -4910.082,E2 -4910.082} C_VEL
LIN {X 0,Y 516.885,Z 452.099,A -85,B 0,C 180,E1 -4910.301,E2 -4910.301} C_VEL
LIN {X 0,Y 516.887,Z 452.099,A -85,B 0,C 180,E1 -4913.342,E2 -4913.342} C_VEL
LIN {X 0,Y 516.915,Z 452.098,A -85,B 0,C 180,E1 -4916.121,E2 -4916.121} C_VEL
LIN {X 0,Y 516.895,Z 452.101,A -85,B 0,C 180,E1 -4918.936,E2 -4918.936} C_VEL
LIN {X 0,Y 516.922,Z 452.094,A -85,B 0,C 180,E1 -4921.585,E2 -4921.585} C_VEL
LIN {X 0,Y 516.936,Z 452.093,A -85,B 0,C 180,E1 -4924.211,E2 -4924.211} C_VEL
LIN {X 0,Y 516.87,Z 452.104,A -85,B 0,C 180,E1 -4926.776,E2 -4926.776} C_VEL
